LIN {X 0,Y 296.94,Z 400.103,A -85,B 0,C 180,E1 -15461.241,E2 -15461.241} C_VEL
LIN {X 0,Y 298.792,Z 385.556,A -85,B 0,C 180,E1 -15462.873,E2 -15462.873} C_VEL
LIN {X 0,Y 295.026,Z 372.369,A -85,B 0,C 180,E1 -15465.675,E2 -15465.675} C_VEL
LIN {X 0,Y 290.73,Z 360.298,A -85,B 0,C 180,E1 -15468.694,E2 -15468.694} C_VEL
LIN {X 0,Y 286.134,Z 349.446,A -85,B 0,C 180,E1 -15471.964,E2 -15471.964} C_VEL
LIN {X 0,Y 282.035,Z 341.18,A -85,B 0,C 180,E1 -15474.962,E2 -15474.962} C_VEL
LIN {X 0,Y 279.846,Z 337.032,A -85,B 0,C 180,E1 -15476.722,E2 -15476.722} C_VEL
LIN {X 0,Y 277.551,Z 332.713,A -85,B 0,C 180,E1 -15478.761,E2 -15478.761} C_VEL
LIN {X 0,Y 275.306,Z 328.719,A -85,B 0,C 180,E1 -15480.832,E2 -15480.832} C_VEL
LIN {X 0,Y 272.385,Z 324.11,A -85,B 0,C 180,E1 -15483.999,E2 -15483.999} C_VEL
LIN {X 0,Y 271.755,Z 322.71,A -85,B 0,C 180,E1 -15484.854,E2 -15484.854} C_VEL
LIN {X 0,Y 268.885,Z 319.004,A -85,B 0,C 180,E1 -15488.984,E2 -15488.984} C_VEL
LIN {X 0,Y 268.106,Z 317.079,A -85,B 0,C 180,E1 -15490.964,E2 -15490.964} C_VEL
LIN {X 0,Y 266.633,Z 315.935,A -85,B 0,C 180,E1 -15497.024,E2 -15497.024} C_VEL
LIN {X 0,Y 267.959,Z 316.873,A -85,B 0,C 180,E1 -15502.891,E2 -15502.891} C_VEL
LIN {X 0,Y 268.11,Z 322.342,A -85,B 0,C 180,E1 -15505.632,E2 -15505.632} C_VEL
LIN {X 0,Y 268.563,Z 325.134,A -85,B 0,C 180,E1 -15506.834,E2 -15506.834} C_VEL
LIN {X 0,Y 280.399,Z 343.647,A -85,B 0,C 180,E1 -15510.42,E2 -15510.42} C_VEL
LIN {X 0,Y 293.861,Z 366.106,A -85,B 0,C 180,E1 -15514.094,E2 -15514.094} C_VEL
LIN {X 0,Y 307.067,Z 389.595,A -85,B 0,C 180,E1 -15517.363,E2 -15517.363} C_VEL
LIN {X 0,Y 311.122,Z 397.45,A -85,B 0,C 180,E1 -15518.324,E2 -15518.324} C_VEL
LIN {X 0,Y 295.469,Z 576.065,A -85,B 0,C 180,E1 -15523.892,E2 -15523.892} C_VEL
LIN {X 0,Y 292.753,Z 597.216,A -85,B 0,C 180,E1 -15524.876,E2 -15524.876} C_VEL
LIN {X 0,Y 289.439,Z 617.893,A -85,B 0,C 180,E1 -15526.18,E2 -15526.18} C_VEL
LIN {X 0,Y 285.489,Z 638.664,A -85,B 0,C 180,E1 -15527.884,E2 -15527.884} C_VEL
LIN {X 0,Y 281.43,Z 657.558,A -85,B 0,C 180,E1 -15529.832,E2 -15529.832} C_VEL
LIN {X 0,Y 277.005,Z 676.334,A -85,B 0,C 180,E1 -15532.23,E2 -15532.23} C_VEL
LIN {X 0,Y 272.656,Z 693.714,A -85,B 0,C 180,E1 -15534.957,E2 -15534.957} C_VEL
LIN {X 0,Y 268.576,Z 709.476,A -85,B 0,C 180,E1 -15537.964,E2 -15537.964} C_VEL
LIN {X 0,Y 264.829,Z 724.067,A -85,B 0,C 180,E1 -15541.351,E2 -15541.351} C_VEL
LIN {X 0,Y 261.74,Z 736.697,A -85,B 0,C 180,E1 -15544.914,E2 -15544.914} C_VEL
LIN {X 0,Y 259.298,Z 747.805,A -85,B 0,C 180,E1 -15548.751,E2 -15548.751} C_VEL
LIN {X 0,Y 257.574,Z 757.323,A -85,B 0,C 180,E1 -15552.844,E2 -15552.844} C_VEL
LIN {X 0,Y 256.562,Z 766.176,A -85,B 0,C 180,E1 -15557.168,E2 -15557.168} C_VEL
LIN {X 0,Y 256.224,Z 771.289,A -85,B 0,C 180,E1 -15560.57,E2 -15560.57} C_VEL
LIN {X 0,Y 256.172,Z 774.841,A -85,B 0,C 180,E1 -15564.178,E2 -15564.178} C_VEL
LIN {X 0,Y 256.225,Z 776.542,A -85,B 0,C 180,E1 -15567.542,E2 -15567.542} C_VEL
LIN {X 0,Y 256.224,Z 776.895,A -85,B 0,C 180,E1 -15571.791,E2 -15571.791} C_VEL
LIN {X 0,Y 256.095,Z 776.47,A -85,B 0,C 180,E1 -15575.604,E2 -15575.604} C_VEL
LIN {X 0,Y 256.135,Z 774.535,A -85,B 0,C 180,E1 -15579.666,E2 -15579.666} C_VEL
LIN {X 0,Y 256.782,Z 770.746,A -85,B 0,C 180,E1 -15584.177,E2 -15584.177} C_VEL
LIN {X 0,Y 258.426,Z 765.131,A -85,B 0,C 180,E1 -15588.734,E2 -15588.734} C_VEL
LIN {X 0,Y 261.437,Z 757.306,A -85,B 0,C 180,E1 -15593.44,E2 -15593.44} C_VEL
LIN {X 0,Y 265.948,Z 747.434,A -85,B 0,C 180,E1 -15598.033,E2 -15598.033} C_VEL
LIN {X 0,Y 272.081,Z 735.449,A -85,B 0,C 180,E1 -15602.45,E2 -15602.45} C_VEL
LIN {X 0,Y 279.493,Z 722.038,A -85,B 0,C 180,E1 -15606.433,E2 -15606.433} C_VEL
LIN {X 0,Y 288.993,Z 705.853,A -85,B 0,C 180,E1 -15610.317,E2 -15610.317} C_VEL
LIN {X 0,Y 299.761,Z 688.525,A -85,B 0,C 180,E1 -15613.668,E2 -15613.668} C_VEL
LIN {X 0,Y 311.664,Z 670.423,A -85,B 0,C 180,E1 -15616.474,E2 -15616.474} C_VEL
LIN {X 0,Y 316.699,Z 662.999,A -85,B 0,C 180,E1 -15617.467,E2 -15617.467} C_VEL
LIN {X 0,Y 304.303,Z 679.759,A -85,B 0,C 180,E1 -15620.155,E2 -15620.155} C_VEL
LIN {X 0,Y 293.114,Z 695.355,A -85,B 0,C 180,E1 -15623.349,E2 -15623.349} C_VEL
LIN {X 0,Y 283.18,Z 709.698,A -85,B 0,C 180,E1 -15627.062,E2 -15627.062} C_VEL
LIN {X 0,Y 275.344,Z 721.405,A -85,B 0,C 180,E1 -15630.884,E2 -15630.884} C_VEL
LIN {X 0,Y 269.011,Z 731.149,A -85,B 0,C 180,E1 -15634.931,E2 -15634.931} C_VEL
LIN {X 0,Y 264.108,Z 738.947,A -85,B 0,C 180,E1 -15639.154,E2 -15639.154} C_VEL
LIN {X 0,Y 260.554,Z 744.818,A -85,B 0,C 180,E1 -15643.503,E2 -15643.503} C_VEL
LIN {X 0,Y 258.222,Z 748.792,A -85,B 0,C 180,E1 -15647.932,E2 -15647.932} C_VEL
LIN {X 0,Y 256.91,Z 750.895,A -85,B 0,C 180,E1 -15652.397,E2 -15652.397} C_VEL
LIN {X 0,Y 256.377,Z 751.195,A -85,B 0,C 180,E1 -15656.423,E2 -15656.423} C_VEL
LIN {X 0,Y 256.196,Z 749.887,A -85,B 0,C 180,E1 -15660.448,E2 -15660.448} C_VEL
LIN {X 0,Y 256.191,Z 747.15,A -85,B 0,C 180,E1 -15664.253,E2 -15664.253} C_VEL
LIN {X 0,Y 256.434,Z 742.885,A -85,B 0,C 180,E1 -15668.07,E2 -15668.07} C_VEL
LIN {X 0,Y 257.125,Z 736.57,A -85,B 0,C 180,E1 -15672.122,E2 -15672.122} C_VEL
LIN {X 0,Y 258.365,Z 728.743,A -85,B 0,C 180,E1 -15675.949,E2 -15675.949} C_VEL
LIN {X 0,Y 260.321,Z 718.846,A -85,B 0,C 180,E1 -15679.773,E2 -15679.773} C_VEL
LIN {X 0,Y 262.858,Z 707.504,A -85,B 0,C 180,E1 -15683.304,E2 -15683.304} C_VEL
LIN {X 0,Y 265.921,Z 694.644,A -85,B 0,C 180,E1 -15686.58,E2 -15686.58} C_VEL
LIN {X 0,Y 269.39,Z 680.327,A -85,B 0,C 180,E1 -15689.581,E2 -15689.581} C_VEL
LIN {X 0,Y 273.303,Z 663.874,A -85,B 0,C 180,E1 -15692.41,E2 -15692.41} C_VEL
LIN {X 0,Y 277.26,Z 646.249,A -85,B 0,C 180,E1 -15694.862,E2 -15694.862} C_VEL
LIN {X 0,Y 281.09,Z 627.597,A -85,B 0,C 180,E1 -15696.953,E2 -15696.953} C_VEL
LIN {X 0,Y 284.671,Z 608.006,A -85,B 0,C 180,E1 -15698.698,E2 -15698.698} C_VEL
LIN {X 0,Y 287.862,Z 587.393,A -85,B 0,C 180,E1 -15700.115,E2 -15700.115} C_VEL
LIN {X 0,Y 290.507,Z 566.391,A -85,B 0,C 180,E1 -15701.175,E2 -15701.175} C_VEL
LIN {X 0,Y 299.392,Z 466.167,A -85,B 0,C 180,E1 -15704.569,E2 -15704.569} C_VEL
LIN {X 0,Y 305.766,Z 396.925,A -85,B 0,C 180,E1 -15706.789,E2 -15706.789} C_VEL
LIN {X 0,Y 293.128,Z 372.457,A -85,B 0,C 180,E1 -15709.952,E2 -15709.952} C_VEL
LIN {X 0,Y 281.063,Z 350.849,A -85,B 0,C 180,E1 -15713.233,E2 -15713.233} C_VEL
LIN {X 0,Y 272.665,Z 336.54,A -85,B 0,C 180,E1 -15715.742,E2 -15715.742} C_VEL
LIN {X 0,Y 271.176,Z 332.651,A -85,B 0,C 180,E1 -15716.965,E2 -15716.965} C_VEL
LIN {X 0,Y 272.605,Z 332.766,A -85,B 0,C 180,E1 -15717.523,E2 -15717.523} C_VEL
LIN {X 0,Y 273.848,Z 333.25,A -85,B 0,C 180,E1 -15717.896,E2 -15717.896} C_VEL
LIN {X 0,Y 279.927,Z 346.608,A -85,B 0,C 180,E1 -15721.25,E2 -15721.25} C_VEL
LIN {X 0,Y 286.015,Z 361.966,A -85,B 0,C 180,E1 -15724.642,E2 -15724.642} C_VEL
LIN {X 0,Y 291.59,Z 378.781,A -85,B 0,C 180,E1 -15727.934,E2 -15727.934} C_VEL
LIN {X 0,Y 292.582,Z 382.952,A -85,B 0,C 180,E1 -15728.655,E2 -15728.655} C_VEL
LIN {X 0,Y 287.272,Z 425.798,A -85,B 0,C 180,E1 -15733.415,E2 -15733.415} C_VEL
LIN {X 0,Y 281.887,Z 470.765,A -85,B 0,C 180,E1 -15738.437,E2 -15738.437} C_VEL
LIN {X 0,Y 280.377,Z 484.638,A -85,B 0,C 180,E1 -15739.986,E2 -15739.986} C_VEL
LIN {X 0,Y 282.331,Z 509.846,A -85,B 0,C 180,E1 -15741.017,E2 -15741.017} C_VEL
LIN {X 0,Y 277.427,Z 629.056,A -85,B 0,C 180,E1 -15744.096,E2 -15744.096} C_VEL
LIN {X 0,Y 276.177,Z 645.328,A -85,B 0,C 180,E1 -15744.896,E2 -15744.896} C_VEL
LIN {X 0,Y 274.405,Z 660.879,A -85,B 0,C 180,E1 -15746.028,E2 -15746.028} C_VEL
LIN {X 0,Y 272.222,Z 675.36,A -85,B 0,C 180,E1 -15747.472,E2 -15747.472} C_VEL
LIN {X 0,Y 269.588,Z 689.834,A -85,B 0,C 180,E1 -15749.36,E2 -15749.36} C_VEL
LIN {X 0,Y 266.915,Z 702.546,A -85,B 0,C 180,E1 -15751.5,E2 -15751.5} C_VEL
LIN {X 0,Y 264.139,Z 714.779,A -85,B 0,C 180,E1 -15754.122,E2 -15754.122} C_VEL
LIN {X 0,Y 261.785,Z 724.548,A -85,B 0,C 180,E1 -15756.797,E2 -15756.797} C_VEL
LIN {X 0,Y 259.615,Z 733.633,A -85,B 0,C 180,E1 -15759.978,E2 -15759.978} C_VEL
LIN {X 0,Y 258.037,Z 740.606,A -85,B 0,C 180,E1 -15763.213,E2 -15763.213} C_VEL
LIN {X 0,Y 256.943,Z 746.215,A -85,B 0,C 180,E1 -15766.806,E2 -15766.806} C_VEL
LIN {X 0,Y 256.412,Z 749.748,A -85,B 0,C 180,E1 -15770.304,E2 -15770.304} C_VEL
LIN {X 0,Y 256.231,Z 751.673,A -85,B 0,C 180,E1 -15774.059,E2 -15774.059} C_VEL
LIN {X 0,Y 256.302,Z 751.729,A -85,B 0,C 180,E1 -15777.657,E2 -15777.657} C_VEL
LIN {X 0,Y 256.718,Z 749.922,A -85,B 0,C 180,E1 -15781.464,E2 -15781.464} C_VEL
LIN {X 0,Y 257.406,Z 747.146,A -85,B 0,C 180,E1 -15784.411,E2 -15784.411} C_VEL
LIN {X 0,Y 256.996,Z 745.207,A -85,B 0,C 180,E1 -15786.083,E2 -15786.083} C_VEL
LIN {X 0,Y 253.978,Z 740.913,A -85,B 0,C 180,E1 -15789.129,E2 -15789.129} C_VEL
LIN {X 0,Y 252.927,Z 737.614,A -85,B 0,C 180,E1 -15790.989,E2 -15790.989} C_VEL
LIN {X 0,Y 253.22,Z 735.69,A -85,B 0,C 180,E1 -15791.898,E2 -15791.898} C_VEL
LIN {X 0,Y 255.85,Z 727.502,A -85,B 0,C 180,E1 -15795.015,E2 -15795.015} C_VEL
LIN {X 0,Y 258.986,Z 717.445,A -85,B 0,C 180,E1 -15797.966,E2 -15797.966} C_VEL
LIN {X 0,Y 262.25,Z 706.223,A -85,B 0,C 180,E1 -15800.534,E2 -15800.534} C_VEL
LIN {X 0,Y 265.744,Z 692.935,A -85,B 0,C 180,E1 -15802.901,E2 -15802.901} C_VEL
LIN {X 0,Y 268.866,Z 679.065,A -85,B 0,C 180,E1 -15804.8,E2 -15804.8} C_VEL
LIN {X 0,Y 271.687,Z 663.938,A -85,B 0,C 180,E1 -15806.376,E2 -15806.376} C_VEL
LIN {X 0,Y 273.868,Z 648.202,A -85,B 0,C 180,E1 -15807.563,E2 -15807.563} C_VEL
LIN {X 0,Y 275.419,Z 631.651,A -85,B 0,C 180,E1 -15808.411,E2 -15808.411} C_VEL
LIN {X 0,Y 278.117,Z 576.528,A -85,B 0,C 180,E1 -15809.917,E2 -15809.917} C_VEL
LIN {X 0,Y 281.382,Z 509.252,A -85,B 0,C 180,E1 -15811.687,E2 -15811.687} C_VEL
LIN {X 0,Y 279.555,Z 485.416,A -85,B 0,C 180,E1 -15812.939,E2 -15812.939} C_VEL
LIN {X 0,Y 285.902,Z 439.143,A -85,B 0,C 180,E1 -15818.132,E2 -15818.132} C_VEL
LIN {X 0,Y 292.228,Z 395.584,A -85,B 0,C 180,E1 -15822.989,E2 -15822.989} C_VEL
LIN {X 0,Y 293.049,Z 389.555,A -85,B 0,C 180,E1 -15823.65,E2 -15823.65} C_VEL
LIN {X 0,Y 289.558,Z 376.947,A -85,B 0,C 180,E1 -15826.419,E2 -15826.419} C_VEL
LIN {X 0,Y 285.465,Z 365.026,A -85,B 0,C 180,E1 -15829.505,E2 -15829.505} C_VEL
LIN {X 0,Y 281.342,Z 355.057,A -85,B 0,C 180,E1 -15832.649,E2 -15832.649} C_VEL
LIN {X 0,Y 277.52,Z 347.06,A -85,B 0,C 180,E1 -15835.66,E2 -15835.66} C_VEL
LIN {X 0,Y 275.656,Z 343.37,A -85,B 0,C 180,E1 -15837.297,E2 -15837.297} C_VEL
LIN {X 0,Y 273.619,Z 339.446,A -85,B 0,C 180,E1 -15839.162,E2 -15839.162} C_VEL
LIN {X 0,Y 271.208,Z 334.904,A -85,B 0,C 180,E1 -15841.689,E2 -15841.689} C_VEL
LIN {X 0,Y 269.01,Z 331.316,A -85,B 0,C 180,E1 -15844.262,E2 -15844.262} C_VEL
LIN {X 0,Y 268.402,Z 329.91,A -85,B 0,C 180,E1 -15845.129,E2 -15845.129} C_VEL
LIN {X 0,Y 265.797,Z 326.228,A -85,B 0,C 180,E1 -15849.308,E2 -15849.308} C_VEL
LIN {X 0,Y 265.181,Z 324.503,A -85,B 0,C 180,E1 -15851.086,E2 -15851.086} C_VEL
LIN {X 0,Y 263.927,Z 323.468,A -85,B 0,C 180,E1 -15857.186,E2 -15857.186} C_VEL
LIN {X 0,Y 265.171,Z 324.337,A -85,B 0,C 180,E1 -15862.519,E2 -15862.519} C_VEL
LIN {X 0,Y 265.167,Z 329.151,A -85,B 0,C 180,E1 -15864.98,E2 -15864.98} C_VEL
LIN {X 0,Y 265.422,Z 332.988,A -85,B 0,C 180,E1 -15866.572,E2 -15866.572} C_VEL
LIN {X 0,Y 277.388,Z 352.176,A -85,B 0,C 180,E1 -15870.306,E2 -15870.306} C_VEL
LIN {X 0,Y 291.163,Z 375.535,A -85,B 0,C 180,E1 -15874.097,E2 -15874.097} C_VEL
LIN {X 0,Y 304.653,Z 399.967,A -85,B 0,C 180,E1 -15877.456,E2 -15877.456} C_VEL
LIN {X 0,Y 288.575,Z 575.961,A -85,B 0,C 180,E1 -15883.096,E2 -15883.096} C_VEL
LIN {X 0,Y 285.646,Z 597.916,A -85,B 0,C 180,E1 -15884.15,E2 -15884.15} C_VEL
LIN {X 0,Y 282.271,Z 618.214,A -85,B 0,C 180,E1 -15885.468,E2 -15885.468} C_VEL
LIN {X 0,Y 278.195,Z 638.944,A -85,B 0,C 180,E1 -15887.216,E2 -15887.216} C_VEL
LIN {X 0,Y 274,Z 657.836,A -85,B 0,C 180,E1 -15889.221,E2 -15889.221} C_VEL
LIN {X 0,Y 269.634,Z 675.826,A -85,B 0,C 180,E1 -15891.573,E2 -15891.573} C_VEL
LIN {X 0,Y 265.139,Z 693.255,A -85,B 0,C 180,E1 -15894.368,E2 -15894.368} C_VEL
LIN {X 0,Y 260.913,Z 709.095,A -85,B 0,C 180,E1 -15897.465,E2 -15897.465} C_VEL
LIN {X 0,Y 257.077,Z 723.582,A -85,B 0,C 180,E1 -15900.914,E2 -15900.914} C_VEL
LIN {X 0,Y 253.884,Z 736.239,A -85,B 0,C 180,E1 -15904.582,E2 -15904.582} C_VEL
LIN {X 0,Y 251.35,Z 747.43,A -85,B 0,C 180,E1 -15908.565,E2 -15908.565} C_VEL
LIN {X 0,Y 249.316,Z 760.034,A -85,B 0,C 180,E1 -15913.699,E2 -15913.699} C_VEL
LIN {X 0,Y 248.554,Z 766.708,A -85,B 0,C 180,E1 -15917.22,E2 -15917.22} C_VEL
LIN {X 0,Y 248.207,Z 771.783,A -85,B 0,C 180,E1 -15920.964,E2 -15920.964} C_VEL
LIN {X 0,Y 248.173,Z 774.842,A -85,B 0,C 180,E1 -15924.454,E2 -15924.454} C_VEL
LIN {X 0,Y 248.24,Z 776.268,A -85,B 0,C 180,E1 -15927.925,E2 -15927.925} C_VEL
LIN {X 0,Y 248.223,Z 776.367,A -85,B 0,C 180,E1 -15932.311,E2 -15932.311} C_VEL
LIN {X 0,Y 248.094,Z 775.911,A -85,B 0,C 180,E1 -15936.249,E2 -15936.249} C_VEL
LIN {X 0,Y 248.218,Z 773.809,A -85,B 0,C 180,E1 -15940.681,E2 -15940.681} C_VEL
LIN {X 0,Y 249.171,Z 769.632,A -85,B 0,C 180,E1 -15945.625,E2 -15945.625} C_VEL
LIN {X 0,Y 251.338,Z 763.593,A -85,B 0,C 180,E1 -15950.494,E2 -15950.494} C_VEL
LIN {X 0,Y 254.987,Z 755.598,A -85,B 0,C 180,E1 -15955.306,E2 -15955.306} C_VEL
LIN {X 0,Y 260.25,Z 745.641,A -85,B 0,C 180,E1 -15959.966,E2 -15959.966} C_VEL
LIN {X 0,Y 267.22,Z 733.705,A -85,B 0,C 180,E1 -15964.404,E2 -15964.404} C_VEL
LIN {X 0,Y 275.965,Z 719.805,A -85,B 0,C 180,E1 -15968.551,E2 -15968.551} C_VEL
LIN {X 0,Y 287.073,Z 703.228,A -85,B 0,C 180,E1 -15972.51,E2 -15972.51} C_VEL
LIN {X 0,Y 299.64,Z 685.661,A -85,B 0,C 180,E1 -15975.845,E2 -15975.845} C_VEL
LIN {X 0,Y 307.526,Z 675.142,A -85,B 0,C 180,E1 -15977.534,E2 -15977.534} C_VEL
LIN {X 0,Y 294.888,Z 690.385,A -85,B 0,C 180,E1 -15980.4,E2 -15980.4} C_VEL
LIN {X 0,Y 282.713,Z 705.662,A -85,B 0,C 180,E1 -15984.088,E2 -15984.088} C_VEL
LIN {X 0,Y 272.716,Z 718.764,A -85,B 0,C 180,E1 -15988.134,E2 -15988.134} C_VEL
LIN {X 0,Y 264.863,Z 729.274,A -85,B 0,C 180,E1 -15992.334,E2 -15992.334} C_VEL
LIN {X 0,Y 258.947,Z 737.428,A -85,B 0,C 180,E1 -15996.566,E2 -15996.566} C_VEL
LIN {X 0,Y 254.487,Z 743.76,A -85,B 0,C 180,E1 -16000.969,E2 -16000.969} C_VEL
LIN {X 0,Y 251.395,Z 748.261,A -85,B 0,C 180,E1 -16005.49,E2 -16005.49} C_VEL
LIN {X 0,Y 249.503,Z 750.937,A -85,B 0,C 180,E1 -16010.078,E2 -16010.078} C_VEL
LIN {X 0,Y 248.594,Z 751.782,A -85,B 0,C 180,E1 -16014.461,E2 -16014.461} C_VEL
LIN {X 0,Y 248.261,Z 751.006,A -85,B 0,C 180,E1 -16018.616,E2 -16018.616} C_VEL
LIN {X 0,Y 248.173,Z 748.831,A -85,B 0,C 180,E1 -16022.541,E2 -16022.541} C_VEL
LIN {X 0,Y 248.31,Z 744.859,A -85,B 0,C 180,E1 -16026.707,E2 -16026.707} C_VEL
LIN {X 0,Y 248.853,Z 739.068,A -85,B 0,C 180,E1 -16030.886,E2 -16030.886} C_VEL
LIN {X 0,Y 250.004,Z 731.303,A -85,B 0,C 180,E1 -16035.069,E2 -16035.069} C_VEL
LIN {X 0,Y 251.806,Z 721.935,A -85,B 0,C 180,E1 -16039.003,E2 -16039.003} C_VEL
LIN {X 0,Y 254.234,Z 711.077,A -85,B 0,C 180,E1 -16042.671,E2 -16042.671} C_VEL
LIN {X 0,Y 257.275,Z 698.511,A -85,B 0,C 180,E1 -16046.133,E2 -16046.133} C_VEL
LIN {X 0,Y 260.864,Z 684.098,A -85,B 0,C 180,E1 -16049.382,E2 -16049.382} C_VEL
LIN {X 0,Y 264.765,Z 668.262,A -85,B 0,C 180,E1 -16052.302,E2 -16052.302} C_VEL
LIN {X 0,Y 268.892,Z 650.709,A -85,B 0,C 180,E1 -16054.936,E2 -16054.936} C_VEL
LIN {X 0,Y 272.949,Z 632.099,A -85,B 0,C 180,E1 -16057.188,E2 -16057.188} C_VEL
LIN {X 0,Y 276.751,Z 612.591,A -85,B 0,C 180,E1 -16059.071,E2 -16059.071} C_VEL
LIN {X 0,Y 280.116,Z 592.33,A -85,B 0,C 180,E1 -16060.583,E2 -16060.583} C_VEL
LIN {X 0,Y 283.01,Z 571.163,A -85,B 0,C 180,E1 -16061.757,E2 -16061.757} C_VEL
LIN {X 0,Y 285.913,Z 541.776,A -85,B 0,C 180,E1 -16062.885,E2 -16062.885} C_VEL
LIN {X 0,Y 299.252,Z 399.79,A -85,B 0,C 180,E1 -16067.637,E2 -16067.637} C_VEL
LIN {X 0,Y 287.388,Z 376.669,A -85,B 0,C 180,E1 -16070.711,E2 -16070.711} C_VEL
LIN {X 0,Y 275.771,Z 355.743,A -85,B 0,C 180,E1 -16073.964,E2 -16073.964} C_VEL
LIN {X 0,Y 266.659,Z 340.131,A -85,B 0,C 180,E1 -16076.806,E2 -16076.806} C_VEL
LIN {X 0,Y 266.891,Z 339.624,A -85,B 0,C 180,E1 -16077.154,E2 -16077.154} C_VEL
LIN {X 0,Y 268.978,Z 339.864,A -85,B 0,C 180,E1 -16077.746,E2 -16077.746} C_VEL
LIN {X 0,Y 275.266,Z 354.159,A -85,B 0,C 180,E1 -16081.347,E2 -16081.347} C_VEL
LIN {X 0,Y 281.019,Z 369.487,A -85,B 0,C 180,E1 -16084.723,E2 -16084.723} C_VEL
LIN {X 0,Y 285.974,Z 385.172,A -85,B 0,C 180,E1 -16087.813,E2 -16087.813} C_VEL
LIN {X 0,Y 281.647,Z 419.515,A -85,B 0,C 180,E1 -16091.687,E2 -16091.687} C_VEL
LIN {X 0,Y 275.942,Z 464.782,A -85,B 0,C 180,E1 -16096.802,E2 -16096.802} C_VEL
LIN {X 0,Y 273.579,Z 484.324,A -85,B 0,C 180,E1 -16099.042,E2 -16099.042} C_VEL
LIN {X 0,Y 275.499,Z 510.719,A -85,B 0,C 180,E1 -16100.17,E2 -16100.17} C_VEL
LIN {X 0,Y 270.405,Z 629.316,A -85,B 0,C 180,E1 -16103.296,E2 -16103.296} C_VEL
LIN {X 0,Y 269.114,Z 645.535,A -85,B 0,C 180,E1 -16104.107,E2 -16104.107} C_VEL
LIN {X 0,Y 267.249,Z 661.287,A -85,B 0,C 180,E1 -16105.276,E2 -16105.276} C_VEL
LIN {X 0,Y 264.975,Z 675.763,A -85,B 0,C 180,E1 -16106.753,E2 -16106.753} C_VEL
LIN {X 0,Y 262.231,Z 690.238,A -85,B 0,C 180,E1 -16108.687,E2 -16108.687} C_VEL
LIN {X 0,Y 259.442,Z 702.948,A -85,B 0,C 180,E1 -16110.881,E2 -16110.881} C_VEL
LIN {X 0,Y 256.54,Z 715.184,A -85,B 0,C 180,E1 -16113.573,E2 -16113.573} C_VEL
LIN {X 0,Y 253.89,Z 725.671,A -85,B 0,C 180,E1 -16116.555,E2 -16116.555} C_VEL
LIN {X 0,Y 251.798,Z 734.038,A -85,B 0,C 180,E1 -16119.598,E2 -16119.598} C_VEL
LIN {X 0,Y 250.137,Z 741.007,A -85,B 0,C 180,E1 -16122.932,E2 -16122.932} C_VEL
LIN {X 0,Y 249.001,Z 746.517,A -85,B 0,C 180,E1 -16126.562,E2 -16126.562} C_VEL
LIN {X 0,Y 248.451,Z 749.972,A -85,B 0,C 180,E1 -16130,E2 -16130} C_VEL
LIN {X 0,Y 248.243,Z 751.951,A -85,B 0,C 180,E1 -16133.749,E2 -16133.749} C_VEL
LIN {X 0,Y 248.296,Z 752.234,A -85,B 0,C 180,E1 -16137.324,E2 -16137.324} C_VEL
LIN {X 0,Y 248.669,Z 750.756,A -85,B 0,C 180,E1 -16141.079,E2 -16141.079} C_VEL
LIN {X 0,Y 249.585,Z 747.388,A -85,B 0,C 180,E1 -16144.947,E2 -16144.947} C_VEL
LIN {X 0,Y 251.035,Z 742.53,A -85,B 0,C 180,E1 -16148.41,E2 -16148.41} C_VEL
LIN {X 0,Y 253.22,Z 735.69,A -85,B 0,C 180,E1 -16151.898,E2 -16151.898} C_VEL
LIN {X 0,Y 253.462,Z 732.181,A -85,B 0,C 180,E1 -16153.464,E2 -16153.464} C_VEL
LIN {X 0,Y 251.407,Z 724.108,A -85,B 0,C 180,E1 -16156.77,E2 -16156.77} C_VEL
LIN {X 0,Y 251.346,Z 719.743,A -85,B 0,C 180,E1 -16158.237,E2 -16158.237} C_VEL
LIN {X 0,Y 251.845,Z 717.662,A -85,B 0,C 180,E1 -16158.823,E2 -16158.823} C_VEL
LIN {X 0,Y 255.273,Z 706.473,A -85,B 0,C 180,E1 -16161.432,E2 -16161.432} C_VEL
LIN {X 0,Y 258.898,Z 693.357,A -85,B 0,C 180,E1 -16163.814,E2 -16163.814} C_VEL
LIN {X 0,Y 262.043,Z 680.108,A -85,B 0,C 180,E1 -16165.674,E2 -16165.674} C_VEL
LIN {X 0,Y 264.995,Z 665.102,A -85,B 0,C 180,E1 -16167.283,E2 -16167.283} C_VEL
LIN {X 0,Y 267.294,Z 649.691,A -85,B 0,C 180,E1 -16168.495,E2 -16168.495} C_VEL
LIN {X 0,Y 268.986,Z 632.949,A -85,B 0,C 180,E1 -16169.39,E2 -16169.39} C_VEL
LIN {X 0,Y 270.617,Z 602.218,A -85,B 0,C 180,E1 -16170.292,E2 -16170.292} C_VEL
LIN {X 0,Y 275.313,Z 510.209,A -85,B 0,C 180,E1 -16172.752,E2 -16172.752} C_VEL
LIN {X 0,Y 273.512,Z 485.979,A -85,B 0,C 180,E1 -16174.058,E2 -16174.058} C_VEL
LIN {X 0,Y 280.045,Z 440.73,A -85,B 0,C 180,E1 -16179.191,E2 -16179.191} C_VEL
LIN {X 0,Y 286.282,Z 399.532,A -85,B 0,C 180,E1 -16183.823,E2 -16183.823} C_VEL
LIN {X 0,Y 287.247,Z 393.097,A -85,B 0,C 180,E1 -16184.556,E2 -16184.556} C_VEL
LIN {X 0,Y 283.992,Z 380.77,A -85,B 0,C 180,E1 -16187.391,E2 -16187.391} C_VEL
LIN {X 0,Y 280.11,Z 369.196,A -85,B 0,C 180,E1 -16190.549,E2 -16190.549} C_VEL
LIN {X 0,Y 275.927,Z 358.91,A -85,B 0,C 180,E1 -16193.967,E2 -16193.967} C_VEL
LIN {X 0,Y 272.236,Z 350.875,A -85,B 0,C 180,E1 -16197.263,E2 -16197.263} C_VEL
LIN {X 0,Y 269.55,Z 345.877,A -85,B 0,C 180,E1 -16199.787,E2 -16199.787} C_VEL
LIN {X 0,Y 267.534,Z 341.803,A -85,B 0,C 180,E1 -16202.141,E2 -16202.141} C_VEL
LIN {X 0,Y 265.369,Z 337.748,A -85,B 0,C 180,E1 -16204.971,E2 -16204.971} C_VEL
LIN {X 0,Y 264.4,Z 336.5,A -85,B 0,C 180,E1 -16206.295,E2 -16206.295} C_VEL
LIN {X 0,Y 262.185,Z 331.841,A -85,B 0,C 180,E1 -16211.437,E2 -16211.437} C_VEL
LIN {X 0,Y 261.185,Z 330.989,A -85,B 0,C 180,E1 -16217.373,E2 -16217.373} C_VEL
LIN {X 0,Y 262.323,Z 331.785,A -85,B 0,C 180,E1 -16222.168,E2 -16222.168} C_VEL
LIN {X 0,Y 262.258,Z 336.015,A -85,B 0,C 180,E1 -16224.338,E2 -16224.338} C_VEL
LIN {X 0,Y 262.325,Z 340.027,A -85,B 0,C 180,E1 -16225.996,E2 -16225.996} C_VEL
LIN {X 0,Y 262.766,Z 341.877,A -85,B 0,C 180,E1 -16226.588,E2 -16226.588} C_VEL
LIN {X 0,Y 275.605,Z 362.845,A -85,B 0,C 180,E1 -16230.554,E2 -16230.554} C_VEL
LIN {X 0,Y 288.747,Z 385.611,A -85,B 0,C 180,E1 -16234.182,E2 -16234.182} C_VEL
LIN {X 0,Y 298.163,Z 403.236,A -85,B 0,C 180,E1 -16236.594,E2 -16236.594} C_VEL
LIN {X 0,Y 281.724,Z 575.658,A -85,B 0,C 180,E1 -16242.265,E2 -16242.265} C_VEL
LIN {X 0,Y 278.71,Z 597.541,A -85,B 0,C 180,E1 -16243.339,E2 -16243.339} C_VEL
LIN {X 0,Y 275.124,Z 618.407,A -85,B 0,C 180,E1 -16244.729,E2 -16244.729} C_VEL
LIN {X 0,Y 270.941,Z 639.009,A -85,B 0,C 180,E1 -16246.513,E2 -16246.513} C_VEL
LIN {X 0,Y 266.524,Z 658.262,A -85,B 0,C 180,E1 -16248.615,E2 -16248.615} C_VEL
LIN {X 0,Y 261.89,Z 676.708,A -85,B 0,C 180,E1 -16251.112,E2 -16251.112} C_VEL
LIN {X 0,Y 257.448,Z 693.416,A -85,B 0,C 180,E1 -16253.882,E2 -16253.882} C_VEL
LIN {X 0,Y 253.07,Z 709.33,A -85,B 0,C 180,E1 -16257.098,E2 -16257.098} C_VEL
LIN {X 0,Y 249.3,Z 723.174,A -85,B 0,C 180,E1 -16260.494,E2 -16260.494} C_VEL
LIN {X 0,Y 246.038,Z 735.711,A -85,B 0,C 180,E1 -16264.229,E2 -16264.229} C_VEL
LIN {X 0,Y 243.824,Z 745.568,A -85,B 0,C 180,E1 -16267.585,E2 -16267.585} C_VEL
LIN {X 0,Y 242.235,Z 754.919,A -85,B 0,C 180,E1 -16270.972,E2 -16270.972} C_VEL
LIN {X 0,Y 241.07,Z 762.731,A -85,B 0,C 180,E1 -16274.609,E2 -16274.609} C_VEL
LIN {X 0,Y 240.415,Z 768.58,A -85,B 0,C 180,E1 -16278.244,E2 -16278.244} C_VEL
LIN {X 0,Y 240.179,Z 772.874,A -85,B 0,C 180,E1 -16282.107,E2 -16282.107} C_VEL
LIN {X 0,Y 240.196,Z 775.247,A -85,B 0,C 180,E1 -16285.706,E2 -16285.706} C_VEL
LIN {X 0,Y 240.275,Z 776.015,A -85,B 0,C 180,E1 -16289.287,E2 -16289.287} C_VEL
LIN {X 0,Y 240.208,Z 775.827,A -85,B 0,C 180,E1 -16293.104,E2 -16293.104} C_VEL
LIN {X 0,Y 240.081,Z 775.292,A -85,B 0,C 180,E1 -16297.18,E2 -16297.18} C_VEL
LIN {X 0,Y 240.332,Z 773.094,A -85,B 0,C 180,E1 -16301.765,E2 -16301.765} C_VEL
LIN {X 0,Y 241.568,Z 768.888,A -85,B 0,C 180,E1 -16306.844,E2 -16306.844} C_VEL
LIN {X 0,Y 244.168,Z 762.817,A -85,B 0,C 180,E1 -16311.881,E2 -16311.881} C_VEL
LIN {X 0,Y 248.363,Z 754.893,A -85,B 0,C 180,E1 -16316.803,E2 -16316.803} C_VEL
LIN {X 0,Y 254.275,Z 745.109,A -85,B 0,C 180,E1 -16321.535,E2 -16321.535} C_VEL
LIN {X 0,Y 262.379,Z 732.889,A -85,B 0,C 180,E1 -16326.207,E2 -16326.207} C_VEL
LIN {X 0,Y 272.493,Z 718.725,A -85,B 0,C 180,E1 -16330.504,E2 -16330.504} C_VEL
LIN {X 0,Y 285.244,Z 702.064,A -85,B 0,C 180,E1 -16334.514,E2 -16334.514} C_VEL
LIN {X 0,Y 298.345,Z 686.007,A -85,B 0,C 180,E1 -16337.582,E2 -16337.582} C_VEL
LIN {X 0,Y 285.435,Z 700.019,A -85,B 0,C 180,E1 -16340.653,E2 -16340.653} C_VEL
LIN {X 0,Y 273.446,Z 713.571,A -85,B 0,C 180,E1 -16344.453,E2 -16344.453} C_VEL
LIN {X 0,Y 263.45,Z 725.221,A -85,B 0,C 180,E1 -16348.672,E2 -16348.672} C_VEL
LIN {X 0,Y 255.57,Z 734.646,A -85,B 0,C 180,E1 -16353.129,E2 -16353.129} C_VEL
LIN {X 0,Y 249.47,Z 742.124,A -85,B 0,C 180,E1 -16357.869,E2 -16357.869} C_VEL
LIN {X 0,Y 245.302,Z 747.328,A -85,B 0,C 180,E1 -16362.52,E2 -16362.52} C_VEL
LIN {X 0,Y 242.619,Z 750.632,A -85,B 0,C 180,E1 -16367.143,E2 -16367.143} C_VEL
LIN {X 0,Y 241.057,Z 752.219,A -85,B 0,C 180,E1 -16371.894,E2 -16371.894} C_VEL
LIN {X 0,Y 240.395,Z 752.015,A -85,B 0,C 180,E1 -16376.424,E2 -16376.424} C_VEL
LIN {X 0,Y 240.2,Z 750.233,A -85,B 0,C 180,E1 -16380.716,E2 -16380.716} C_VEL
LIN {X 0,Y 240.21,Z 747.067,A -85,B 0,C 180,E1 -16384.776,E2 -16384.776} C_VEL
LIN {X 0,Y 240.52,Z 742.34,A -85,B 0,C 180,E1 -16388.849,E2 -16388.849} C_VEL
LIN {X 0,Y 241.371,Z 735.455,A -85,B 0,C 180,E1 -16393.17,E2 -16393.17} C_VEL
LIN {X 0,Y 242.857,Z 727.042,A -85,B 0,C 180,E1 -16397.244,E2 -16397.244} C_VEL
LIN {X 0,Y 244.974,Z 717.208,A -85,B 0,C 180,E1 -16401.05,E2 -16401.05} C_VEL
LIN {X 0,Y 247.871,Z 705.176,A -85,B 0,C 180,E1 -16404.82,E2 -16404.82} C_VEL
LIN {X 0,Y 251.297,Z 691.714,A -85,B 0,C 180,E1 -16408.261,E2 -16408.261} C_VEL
LIN {X 0,Y 255.157,Z 676.643,A -85,B 0,C 180,E1 -16411.412,E2 -16411.412} C_VEL
LIN {X 0,Y 259.477,Z 659.25,A -85,B 0,C 180,E1 -16414.37,E2 -16414.37} C_VEL
LIN {X 0,Y 263.643,Z 641.466,A -85,B 0,C 180,E1 -16416.814,E2 -16416.814} C_VEL
LIN {X 0,Y 267.756,Z 622.179,A -85,B 0,C 180,E1 -16418.945,E2 -16418.945} C_VEL
LIN {X 0,Y 271.494,Z 602.071,A -85,B 0,C 180,E1 -16420.683,E2 -16420.683} C_VEL
LIN {X 0,Y 274.769,Z 581.052,A -85,B 0,C 180,E1 -16422.064,E2 -16422.064} C_VEL
LIN {X 0,Y 277.472,Z 558.924,A -85,B 0,C 180,E1 -16423.104,E2 -16423.104} C_VEL
LIN {X 0,Y 292.736,Z 402.476,A -85,B 0,C 180,E1 -16428.531,E2 -16428.531} C_VEL
LIN {X 0,Y 280.402,Z 378.491,A -85,B 0,C 180,E1 -16431.844,E2 -16431.844} C_VEL
LIN {X 0,Y 268.661,Z 357.396,A -85,B 0,C 180,E1 -16435.289,E2 -16435.289} C_VEL
LIN {X 0,Y 263.05,Z 347.539,A -85,B 0,C 180,E1 -16437.145,E2 -16437.145} C_VEL
LIN {X 0,Y 263.382,Z 346.943,A -85,B 0,C 180,E1 -16437.435,E2 -16437.435} C_VEL
LIN {X 0,Y 264.367,Z 347.015,A -85,B 0,C 180,E1 -16437.726,E2 -16437.726} C_VEL
LIN {X 0,Y 270.486,Z 361.582,A -85,B 0,C 180,E1 -16441.395,E2 -16441.395} C_VEL
LIN {X 0,Y 276.098,Z 377.318,A -85,B 0,C 180,E1 -16444.872,E2 -16444.872} C_VEL
LIN {X 0,Y 279.437,Z 389.009,A -85,B 0,C 180,E1 -16447.154,E2 -16447.154} C_VEL
LIN {X 0,Y 273.666,Z 431.774,A -85,B 0,C 180,E1 -16452.015,E2 -16452.015} C_VEL
LIN {X 0,Y 267.938,Z 475.725,A -85,B 0,C 180,E1 -16457.06,E2 -16457.06} C_VEL
LIN {X 0,Y 266.869,Z 485.441,A -85,B 0,C 180,E1 -16458.147,E2 -16458.147} C_VEL
LIN {X 0,Y 268.738,Z 511.464,A -85,B 0,C 180,E1 -16459.277,E2 -16459.277} C_VEL
LIN {X 0,Y 263.4,Z 629.84,A -85,B 0,C 180,E1 -16462.473,E2 -16462.473} C_VEL
LIN {X 0,Y 262.031,Z 646.203,A -85,B 0,C 180,E1 -16463.314,E2 -16463.314} C_VEL
LIN {X 0,Y 260.134,Z 661.581,A -85,B 0,C 180,E1 -16464.484,E2 -16464.484} C_VEL
LIN {X 0,Y 257.767,Z 676.09,A -85,B 0,C 180,E1 -16465.994,E2 -16465.994} C_VEL
LIN {X 0,Y 254.908,Z 690.584,A -85,B 0,C 180,E1 -16467.975,E2 -16467.975} C_VEL
LIN {X 0,Y 251.971,Z 703.426,A -85,B 0,C 180,E1 -16470.248,E2 -16470.248} C_VEL
LIN {X 0,Y 248.964,Z 715.561,A -85,B 0,C 180,E1 -16472.99,E2 -16472.99} C_VEL
LIN {X 0,Y 246.29,Z 725.681,A -85,B 0,C 180,E1 -16475.934,E2 -16475.934} C_VEL
LIN {X 0,Y 243.991,Z 734.43,A -85,B 0,C 180,E1 -16479.194,E2 -16479.194} C_VEL
LIN {X 0,Y 242.244,Z 741.402,A -85,B 0,C 180,E1 -16482.633,E2 -16482.633} C_VEL
LIN {X 0,Y 241.046,Z 746.913,A -85,B 0,C 180,E1 -16486.381,E2 -16486.381} C_VEL
LIN {X 0,Y 240.46,Z 750.406,A -85,B 0,C 180,E1 -16489.99,E2 -16489.99} C_VEL
LIN {X 0,Y 240.251,Z 752.346,A -85,B 0,C 180,E1 -16493.806,E2 -16493.806} C_VEL
LIN {X 0,Y 240.321,Z 752.618,A -85,B 0,C 180,E1 -16497.599,E2 -16497.599} C_VEL
LIN {X 0,Y 240.756,Z 751.048,A -85,B 0,C 180,E1 -16501.549,E2 -16501.549} C_VEL
LIN {X 0,Y 241.757,Z 747.721,A -85,B 0,C 180,E1 -16505.435,E2 -16505.435} C_VEL
LIN {X 0,Y 243.459,Z 742.459,A -85,B 0,C 180,E1 -16509.228,E2 -16509.228} C_VEL
LIN {X 0,Y 245.836,Z 735.559,A -85,B 0,C 180,E1 -16512.778,E2 -16512.778} C_VEL
LIN {X 0,Y 248.868,Z 726.664,A -85,B 0,C 180,E1 -16516.158,E2 -16516.158} C_VEL
LIN {X 0,Y 251.845,Z 717.662,A -85,B 0,C 180,E1 -16518.823,E2 -16518.823} C_VEL
LIN {X 0,Y 252.569,Z 712.778,A -85,B 0,C 180,E1 -16520.187,E2 -16520.187} C_VEL
LIN {X 0,Y 251.472,Z 702.771,A -85,B 0,C 180,E1 -16522.915,E2 -16522.915} C_VEL
LIN {X 0,Y 251.596,Z 696.374,A -85,B 0,C 180,E1 -16524.323,E2 -16524.323} C_VEL
LIN {X 0,Y 252.14,Z 693.786,A -85,B 0,C 180,E1 -16524.782,E2 -16524.782} C_VEL
LIN {X 0,Y 255.515,Z 680.254,A -85,B 0,C 180,E1 -16526.716,E2 -16526.716} C_VEL
LIN {X 0,Y 258.516,Z 665.707,A -85,B 0,C 180,E1 -16528.303,E2 -16528.303} C_VEL
LIN {X 0,Y 260.934,Z 650.295,A -85,B 0,C 180,E1 -16529.54,E2 -16529.54} C_VEL
LIN {X 0,Y 262.727,Z 633.392,A -85,B 0,C 180,E1 -16530.46,E2 -16530.46} C_VEL
LIN {X 0,Y 264.426,Z 602.955,A -85,B 0,C 180,E1 -16531.369,E2 -16531.369} C_VEL
LIN {X 0,Y 269.357,Z 511.316,A -85,B 0,C 180,E1 -16533.859,E2 -16533.859} C_VEL
LIN {X 0,Y 267.623,Z 486.252,A -85,B 0,C 180,E1 -16535.263,E2 -16535.263} C_VEL
LIN {X 0,Y 274.663,Z 440.447,A -85,B 0,C 180,E1 -16540.525,E2 -16540.525} C_VEL
LIN {X 0,Y 281.678,Z 396.905,A -85,B 0,C 180,E1 -16545.481,E2 -16545.481} C_VEL
LIN {X 0,Y 278.503,Z 384.661,A -85,B 0,C 180,E1 -16548.401,E2 -16548.401} C_VEL
LIN {X 0,Y 275.112,Z 374.138,A -85,B 0,C 180,E1 -16551.43,E2 -16551.43} C_VEL
LIN {X 0,Y 271.329,Z 364.565,A -85,B 0,C 180,E1 -16554.713,E2 -16554.713} C_VEL
LIN {X 0,Y 268.101,Z 357.243,A -85,B 0,C 180,E1 -16557.862,E2 -16557.862} C_VEL
LIN {X 0,Y 265.809,Z 352.672,A -85,B 0,C 180,E1 -16560.215,E2 -16560.215} C_VEL
LIN {X 0,Y 264.137,Z 348.957,A -85,B 0,C 180,E1 -16562.386,E2 -16562.386} C_VEL
LIN {X 0,Y 262.032,Z 344.964,A -85,B 0,C 180,E1 -16565.254,E2 -16565.254} C_VEL
LIN {X 0,Y 261.21,Z 343.736,A -85,B 0,C 180,E1 -16566.593,E2 -16566.593} C_VEL
LIN {X 0,Y 259.249,Z 339.266,A -85,B 0,C 180,E1 -16571.605,E2 -16571.605} C_VEL
LIN {X 0,Y 258.446,Z 338.509,A -85,B 0,C 180,E1 -16577.563,E2 -16577.563} C_VEL
LIN {X 0,Y 259.489,Z 339.421,A -85,B 0,C 180,E1 -16581.947,E2 -16581.947} C_VEL
LIN {X 0,Y 259.379,Z 345.514,A -85,B 0,C 180,E1 -16584.845,E2 -16584.845} C_VEL
LIN {X 0,Y 259.573,Z 350.003,A -85,B 0,C 180,E1 -16586.385,E2 -16586.385} C_VEL
LIN {X 0,Y 271.338,Z 369.415,A -85,B 0,C 180,E1 -16590.075,E2 -16590.075} C_VEL
LIN {X 0,Y 283.805,Z 391.256,A -85,B 0,C 180,E1 -16593.611,E2 -16593.611} C_VEL
LIN {X 0,Y 291.694,Z 406.109,A -85,B 0,C 180,E1 -16595.695,E2 -16595.695} C_VEL
LIN {X 0,Y 274.876,Z 575.506,A -85,B 0,C 180,E1 -16601.413,E2 -16601.413} C_VEL
LIN {X 0,Y 271.832,Z 596.932,A -85,B 0,C 180,E1 -16602.487,E2 -16602.487} C_VEL
LIN {X 0,Y 268.025,Z 618.404,A -85,B 0,C 180,E1 -16603.951,E2 -16603.951} C_VEL
LIN {X 0,Y 263.729,Z 638.906,A -85,B 0,C 180,E1 -16605.77,E2 -16605.77} C_VEL
LIN {X 0,Y 259.299,Z 657.672,A -85,B 0,C 180,E1 -16607.864,E2 -16607.864} C_VEL
LIN {X 0,Y 254.654,Z 675.677,A -85,B 0,C 180,E1 -16610.344,E2 -16610.344} C_VEL
LIN {X 0,Y 249.995,Z 692.7,A -85,B 0,C 180,E1 -16613.221,E2 -16613.221} C_VEL
LIN {X 0,Y 245.488,Z 708.606,A -85,B 0,C 180,E1 -16616.507,E2 -16616.507} C_VEL
LIN {X 0,Y 241.388,Z 723.196,A -85,B 0,C 180,E1 -16620.198,E2 -16620.198} C_VEL
LIN {X 0,Y 238.102,Z 736.125,A -85,B 0,C 180,E1 -16623.979,E2 -16623.979} C_VEL
LIN {X 0,Y 235.984,Z 746.974,A -85,B 0,C 180,E1 -16627.324,E2 -16627.324} C_VEL
LIN {X 0,Y 234.301,Z 755.943,A -85,B 0,C 180,E1 -16630.82,E2 -16630.82} C_VEL
LIN {X 0,Y 233.077,Z 763.404,A -85,B 0,C 180,E1 -16634.578,E2 -16634.578} C_VEL
LIN {X 0,Y 232.378,Z 769.258,A -85,B 0,C 180,E1 -16638.587,E2 -16638.587} C_VEL
LIN {X 0,Y 232.172,Z 772.992,A -85,B 0,C 180,E1 -16642.331,E2 -16642.331} C_VEL
LIN {X 0,Y 232.21,Z 775.067,A -85,B 0,C 180,E1 -16646.052,E2 -16646.052} C_VEL
LIN {X 0,Y 232.292,Z 775.579,A -85,B 0,C 180,E1 -16649.756,E2 -16649.756} C_VEL
LIN {X 0,Y 232.233,Z 775.277,A -85,B 0,C 180,E1 -16652.964,E2 -16652.964} C_VEL
LIN {X 0,Y 232.091,Z 774.894,A -85,B 0,C 180,E1 -16657.18,E2 -16657.18} C_VEL
LIN {X 0,Y 232.348,Z 773.008,A -85,B 0,C 180,E1 -16661.923,E2 -16661.923} C_VEL
LIN {X 0,Y 233.577,Z 769.389,A -85,B 0,C 180,E1 -16666.925,E2 -16666.925} C_VEL
LIN {X 0,Y 236.446,Z 763.468,A -85,B 0,C 180,E1 -16672.372,E2 -16672.372} C_VEL
LIN {X 0,Y 241.157,Z 755.58,A -85,B 0,C 180,E1 -16677.671,E2 -16677.671} C_VEL
LIN {X 0,Y 248.196,Z 745.291,A -85,B 0,C 180,E1 -16682.949,E2 -16682.949} C_VEL
LIN {X 0,Y 257.447,Z 732.968,A -85,B 0,C 180,E1 -16687.855,E2 -16687.855} C_VEL
LIN {X 0,Y 269.502,Z 718.104,A -85,B 0,C 180,E1 -16692.474,E2 -16692.474} C_VEL
LIN {X 0,Y 283.352,Z 702.222,A -85,B 0,C 180,E1 -16696.337,E2 -16696.337} C_VEL
LIN {X 0,Y 289.035,Z 696.015,A -85,B 0,C 180,E1 -16697.647,E2 -16697.647} C_VEL
LIN {X 0,Y 275.346,Z 709.401,A -85,B 0,C 180,E1 -16701.083,E2 -16701.083} C_VEL
LIN {X 0,Y 263.037,Z 721.802,A -85,B 0,C 180,E1 -16705.238,E2 -16705.238} C_VEL
LIN {X 0,Y 252.946,Z 732.321,A -85,B 0,C 180,E1 -16709.868,E2 -16709.868} C_VEL
LIN {X 0,Y 245.312,Z 740.47,A -85,B 0,C 180,E1 -16714.662,E2 -16714.662} C_VEL
LIN {X 0,Y 239.818,Z 746.395,A -85,B 0,C 180,E1 -16719.5,E2 -16719.5} C_VEL
LIN {X 0,Y 236.002,Z 750.456,A -85,B 0,C 180,E1 -16724.52,E2 -16724.52} C_VEL
LIN {X 0,Y 233.765,Z 752.545,A -85,B 0,C 180,E1 -16729.403,E2 -16729.403} C_VEL
LIN {X 0,Y 232.675,Z 752.869,A -85,B 0,C 180,E1 -16734.081,E2 -16734.081} C_VEL
LIN {X 0,Y 232.274,Z 751.624,A -85,B 0,C 180,E1 -16738.521,E2 -16738.521} C_VEL
LIN {X 0,Y 232.176,Z 749.013,A -85,B 0,C 180,E1 -16742.716,E2 -16742.716} C_VEL
LIN {X 0,Y 232.325,Z 744.909,A -85,B 0,C 180,E1 -16746.922,E2 -16746.922} C_VEL
LIN {X 0,Y 232.887,Z 739.168,A -85,B 0,C 180,E1 -16751.141,E2 -16751.141} C_VEL
LIN {X 0,Y 234.051,Z 731.644,A -85,B 0,C 180,E1 -16755.36,E2 -16755.36} C_VEL
LIN {X 0,Y 235.982,Z 722.115,A -85,B 0,C 180,E1 -16759.557,E2 -16759.557} C_VEL
LIN {X 0,Y 238.593,Z 711.091,A -85,B 0,C 180,E1 -16763.461,E2 -16763.461} C_VEL
LIN {X 0,Y 241.789,Z 698.652,A -85,B 0,C 180,E1 -16767.058,E2 -16767.058} C_VEL
LIN {X 0,Y 245.586,Z 684.276,A -85,B 0,C 180,E1 -16770.457,E2 -16770.457} C_VEL
LIN {X 0,Y 249.754,Z 668.328,A -85,B 0,C 180,E1 -16773.537,E2 -16773.537} C_VEL
LIN {X 0,Y 254.158,Z 650.692,A -85,B 0,C 180,E1 -16776.305,E2 -16776.305} C_VEL
LIN {X 0,Y 258.477,Z 632.032,A -85,B 0,C 180,E1 -16778.663,E2 -16778.663} C_VEL
LIN {X 0,Y 262.541,Z 612.369,A -85,B 0,C 180,E1 -16780.636,E2 -16780.636} C_VEL
LIN {X 0,Y 266.041,Z 592.568,A -85,B 0,C 180,E1 -16782.179,E2 -16782.179} C_VEL
LIN {X 0,Y 269.162,Z 571.164,A -85,B 0,C 180,E1 -16783.421,E2 -16783.421} C_VEL
LIN {X 0,Y 272.248,Z 542.164,A -85,B 0,C 180,E1 -16784.592,E2 -16784.592} C_VEL
LIN {X 0,Y 286.213,Z 405.215,A -85,B 0,C 180,E1 -16789.439,E2 -16789.439} C_VEL
LIN {X 0,Y 274.152,Z 381.732,A -85,B 0,C 180,E1 -16792.804,E2 -16792.804} C_VEL
LIN {X 0,Y 263.313,Z 362.162,A -85,B 0,C 180,E1 -16796.1,E2 -16796.1} C_VEL
LIN {X 0,Y 259.462,Z 355.12,A -85,B 0,C 180,E1 -16797.456,E2 -16797.456} C_VEL
LIN {X 0,Y 259.948,Z 354.608,A -85,B 0,C 180,E1 -16797.803,E2 -16797.803} C_VEL
LIN {X 0,Y 265.947,Z 369.757,A -85,B 0,C 180,E1 -16801.614,E2 -16801.614} C_VEL
LIN {X 0,Y 270.932,Z 384.639,A -85,B 0,C 180,E1 -16804.885,E2 -16804.885} C_VEL
LIN {X 0,Y 272.965,Z 392.002,A -85,B 0,C 180,E1 -16806.34,E2 -16806.34} C_VEL
LIN {X 0,Y 267.1,Z 433.334,A -85,B 0,C 180,E1 -16811.105,E2 -16811.105} C_VEL
LIN {X 0,Y 261.43,Z 474.987,A -85,B 0,C 180,E1 -16815.942,E2 -16815.942} C_VEL
LIN {X 0,Y 260.198,Z 485.826,A -85,B 0,C 180,E1 -16817.164,E2 -16817.164} C_VEL
LIN {X 0,Y 262.028,Z 512.289,A -85,B 0,C 180,E1 -16818.344,E2 -16818.344} C_VEL
LIN {X 0,Y 256.451,Z 630.322,A -85,B 0,C 180,E1 -16821.605,E2 -16821.605} C_VEL
LIN {X 0,Y 255.011,Z 646.741,A -85,B 0,C 180,E1 -16822.471,E2 -16822.471} C_VEL
LIN {X 0,Y 253.07,Z 661.849,A -85,B 0,C 180,E1 -16823.646,E2 -16823.646} C_VEL
LIN {X 0,Y 250.605,Z 676.391,A -85,B 0,C 180,E1 -16825.191,E2 -16825.191} C_VEL
LIN {X 0,Y 247.624,Z 690.905,A -85,B 0,C 180,E1 -16827.22,E2 -16827.22} C_VEL
LIN {X 0,Y 244.589,Z 703.65,A -85,B 0,C 180,E1 -16829.529,E2 -16829.529} C_VEL
LIN {X 0,Y 241.413,Z 715.913,A -85,B 0,C 180,E1 -16832.371,E2 -16832.371} C_VEL
LIN {X 0,Y 238.505,Z 726.419,A -85,B 0,C 180,E1 -16835.53,E2 -16835.53} C_VEL
LIN {X 0,Y 236.196,Z 734.801,A -85,B 0,C 180,E1 -16838.763,E2 -16838.763} C_VEL
LIN {X 0,Y 234.356,Z 741.78,A -85,B 0,C 180,E1 -16842.314,E2 -16842.314} C_VEL
LIN {X 0,Y 233.093,Z 747.297,A -85,B 0,C 180,E1 -16846.187,E2 -16846.187} C_VEL
LIN {X 0,Y 232.482,Z 750.755,A -85,B 0,C 180,E1 -16849.859,E2 -16849.859} C_VEL
LIN {X 0,Y 232.258,Z 752.739,A -85,B 0,C 180,E1 -16853.867,E2 -16853.867} C_VEL
LIN {X 0,Y 232.336,Z 753.025,A -85,B 0,C 180,E1 -16857.692,E2 -16857.692} C_VEL
LIN {X 0,Y 232.802,Z 751.526,A -85,B 0,C 180,E1 -16861.744,E2 -16861.744} C_VEL
LIN {X 0,Y 233.903,Z 748.174,A -85,B 0,C 180,E1 -16865.844,E2 -16865.844} C_VEL
LIN {X 0,Y 235.607,Z 743.314,A -85,B 0,C 180,E1 -16869.532,E2 -16869.532} C_VEL
LIN {X 0,Y 238.092,Z 736.561,A -85,B 0,C 180,E1 -16873.193,E2 -16873.193} C_VEL
LIN {X 0,Y 241.11,Z 728.302,A -85,B 0,C 180,E1 -16876.523,E2 -16876.523} C_VEL
LIN {X 0,Y 244.661,Z 718.184,A -85,B 0,C 180,E1 -16879.647,E2 -16879.647} C_VEL
LIN {X 0,Y 248.154,Z 707.442,A -85,B 0,C 180,E1 -16882.233,E2 -16882.233} C_VEL
LIN {X 0,Y 251.913,Z 694.598,A -85,B 0,C 180,E1 -16884.645,E2 -16884.645} C_VEL
LIN {X 0,Y 252.14,Z 693.786,A -85,B 0,C 180,E1 -16884.782,E2 -16884.782} C_VEL
LIN {X 0,Y 252.943,Z 687.682,A -85,B 0,C 180,E1 -16885.858,E2 -16885.858} C_VEL
LIN {X 0,Y 251.847,Z 673.719,A -85,B 0,C 180,E1 -16888.384,E2 -16888.384} C_VEL
LIN {X 0,Y 252.061,Z 667.063,A -85,B 0,C 180,E1 -16889.289,E2 -16889.289} C_VEL
LIN {X 0,Y 252.375,Z 665.07,A -85,B 0,C 180,E1 -16889.497,E2 -16889.497} C_VEL
LIN {X 0,Y 254.891,Z 649.347,A -85,B 0,C 180,E1 -16890.743,E2 -16890.743} C_VEL
LIN {X 0,Y 256.676,Z 632.86,A -85,B 0,C 180,E1 -16891.631,E2 -16891.631} C_VEL
LIN {X 0,Y 260.161,Z 572.117,A -85,B 0,C 180,E1 -16893.376,E2 -16893.376} C_VEL
LIN {X 0,Y 263.538,Z 512.271,A -85,B 0,C 180,E1 -16895.032,E2 -16895.032} C_VEL
LIN {X 0,Y 261.859,Z 487.034,A -85,B 0,C 180,E1 -16896.483,E2 -16896.483} C_VEL
LIN {X 0,Y 269.118,Z 441.982,A -85,B 0,C 180,E1 -16901.702,E2 -16901.702} C_VEL
LIN {X 0,Y 276.117,Z 400.724,A -85,B 0,C 180,E1 -16906.439,E2 -16906.439} C_VEL
LIN {X 0,Y 273.39,Z 389.42,A -85,B 0,C 180,E1 -16909.249,E2 -16909.249} C_VEL
LIN {X 0,Y 270.594,Z 380.2,A -85,B 0,C 180,E1 -16911.98,E2 -16911.98} C_VEL
LIN {X 0,Y 267.148,Z 370.865,A -85,B 0,C 180,E1 -16915.276,E2 -16915.276} C_VEL
LIN {X 0,Y 264.039,Z 363.618,A -85,B 0,C 180,E1 -16918.48,E2 -16918.48} C_VEL
LIN {X 0,Y 262.156,Z 359.505,A -85,B 0,C 180,E1 -16920.655,E2 -16920.655} C_VEL
LIN {X 0,Y 260.523,Z 355.857,A -85,B 0,C 180,E1 -16922.859,E2 -16922.859} C_VEL
LIN {X 0,Y 258.425,Z 351.439,A -85,B 0,C 180,E1 -16926.218,E2 -16926.218} C_VEL
LIN {X 0,Y 256.516,Z 347.354,A -85,B 0,C 180,E1 -16930.827,E2 -16930.827} C_VEL
LIN {X 0,Y 256.252,Z 346.625,A -85,B 0,C 180,E1 -16932.163,E2 -16932.163} C_VEL
LIN {X 0,Y 255.772,Z 346.054,A -85,B 0,C 180,E1 -16937.752,E2 -16937.752} C_VEL
LIN {X 0,Y 256.678,Z 346.655,A -85,B 0,C 180,E1 -16941.479,E2 -16941.479} C_VEL
LIN {X 0,Y 256.428,Z 352.391,A -85,B 0,C 180,E1 -16944.167,E2 -16944.167} C_VEL
LIN {X 0,Y 256.52,Z 358.28,A -85,B 0,C 180,E1 -16946.225,E2 -16946.225} C_VEL
LIN {X 0,Y 268.181,Z 377.95,A -85,B 0,C 180,E1 -16949.941,E2 -16949.941} C_VEL
LIN {X 0,Y 280.331,Z 399.558,A -85,B 0,C 180,E1 -16953.427,E2 -16953.427} C_VEL
LIN {X 0,Y 285.231,Z 409.114,A -85,B 0,C 180,E1 -16954.772,E2 -16954.772} C_VEL
LIN {X 0,Y 268.013,Z 575.619,A -85,B 0,C 180,E1 -16960.546,E2 -16960.546} C_VEL
LIN {X 0,Y 264.884,Z 596.863,A -85,B 0,C 180,E1 -16961.64,E2 -16961.64} C_VEL
LIN {X 0,Y 260.978,Z 618.204,A -85,B 0,C 180,E1 -16963.131,E2 -16963.131} C_VEL
LIN {X 0,Y 256.566,Z 638.64,A -85,B 0,C 180,E1 -16964.987,E2 -16964.987} C_VEL
LIN {X 0,Y 251.791,Z 658.206,A -85,B 0,C 180,E1 -16967.235,E2 -16967.235} C_VEL
LIN {X 0,Y 247.008,Z 676.133,A -85,B 0,C 180,E1 -16969.791,E2 -16969.791} C_VEL
LIN {X 0,Y 242.353,Z 692.634,A -85,B 0,C 180,E1 -16972.669,E2 -16972.669} C_VEL
LIN {X 0,Y 237.684,Z 708.623,A -85,B 0,C 180,E1 -16976.082,E2 -16976.082} C_VEL
LIN {X 0,Y 233.255,Z 724.496,A -85,B 0,C 180,E1 -16980.111,E2 -16980.111} C_VEL
LIN {X 0,Y 230.681,Z 736.731,A -85,B 0,C 180,E1 -16983.236,E2 -16983.236} C_VEL
LIN {X 0,Y 228.298,Z 747.641,A -85,B 0,C 180,E1 -16986.789,E2 -16986.789} C_VEL
LIN {X 0,Y 226.476,Z 756.403,A -85,B 0,C 180,E1 -16990.399,E2 -16990.399} C_VEL
LIN {X 0,Y 225.149,Z 763.621,A -85,B 0,C 180,E1 -16994.286,E2 -16994.286} C_VEL
LIN {X 0,Y 224.392,Z 769.313,A -85,B 0,C 180,E1 -16998.436,E2 -16998.436} C_VEL
LIN {X 0,Y 224.168,Z 773.013,A -85,B 0,C 180,E1 -17002.571,E2 -17002.571} C_VEL
LIN {X 0,Y 224.224,Z 774.858,A -85,B 0,C 180,E1 -17006.424,E2 -17006.424} C_VEL
LIN {X 0,Y 224.304,Z 775.142,A -85,B 0,C 180,E1 -17010.258,E2 -17010.258} C_VEL
LIN {X 0,Y 224.239,Z 774.681,A -85,B 0,C 180,E1 -17013.326,E2 -17013.326} C_VEL
LIN {X 0,Y 224.104,Z 774.334,A -85,B 0,C 180,E1 -17017.953,E2 -17017.953} C_VEL
LIN {X 0,Y 224.526,Z 772.338,A -85,B 0,C 180,E1 -17023.13,E2 -17023.13} C_VEL
LIN {X 0,Y 226.218,Z 768.472,A -85,B 0,C 180,E1 -17028.559,E2 -17028.559} C_VEL
LIN {X 0,Y 229.7,Z 762.535,A -85,B 0,C 180,E1 -17034.155,E2 -17034.155} C_VEL
LIN {X 0,Y 235.455,Z 754.321,A -85,B 0,C 180,E1 -17039.794,E2 -17039.794} C_VEL
LIN {X 0,Y 243.487,Z 744.149,A -85,B 0,C 180,E1 -17045.095,E2 -17045.095} C_VEL
LIN {X 0,Y 254.295,Z 731.59,A -85,B 0,C 180,E1 -17050.155,E2 -17050.155} C_VEL
LIN {X 0,Y 267.584,Z 717.288,A -85,B 0,C 180,E1 -17054.629,E2 -17054.629} C_VEL
LIN {X 0,Y 279.674,Z 705.089,A -85,B 0,C 180,E1 -17057.701,E2 -17057.701} C_VEL
LIN {X 0,Y 265.174,Z 717.754,A -85,B 0,C 180,E1 -17061.528,E2 -17061.528} C_VEL
LIN {X 0,Y 252.612,Z 729.11,A -85,B 0,C 180,E1 -17066.077,E2 -17066.077} C_VEL
LIN {X 0,Y 242.853,Z 738.169,A -85,B 0,C 180,E1 -17070.934,E2 -17070.934} C_VEL
LIN {X 0,Y 235.58,Z 744.978,A -85,B 0,C 180,E1 -17075.956,E2 -17075.956} C_VEL
LIN {X 0,Y 230.269,Z 749.837,A -85,B 0,C 180,E1 -17081.258,E2 -17081.258} C_VEL
LIN {X 0,Y 226.95,Z 752.62,A -85,B 0,C 180,E1 -17086.498,E2 -17086.498} C_VEL
LIN {X 0,Y 225.16,Z 753.534,A -85,B 0,C 180,E1 -17091.574,E2 -17091.574} C_VEL
LIN {X 0,Y 224.408,Z 752.743,A -85,B 0,C 180,E1 -17096.447,E2 -17096.447} C_VEL
LIN {X 0,Y 224.198,Z 750.439,A -85,B 0,C 180,E1 -17101.023,E2 -17101.023} C_VEL
LIN {X 0,Y 224.234,Z 746.715,A -85,B 0,C 180,E1 -17105.374,E2 -17105.374} C_VEL
LIN {X 0,Y 224.634,Z 741.414,A -85,B 0,C 180,E1 -17109.739,E2 -17109.739} C_VEL
LIN {X 0,Y 225.605,Z 734.39,A -85,B 0,C 180,E1 -17114.109,E2 -17114.109} C_VEL
LIN {X 0,Y 227.332,Z 725.447,A -85,B 0,C 180,E1 -17118.463,E2 -17118.463} C_VEL
LIN {X 0,Y 229.76,Z 715.051,A -85,B 0,C 180,E1 -17122.518,E2 -17122.518} C_VEL
LIN {X 0,Y 232.803,Z 703.296,A -85,B 0,C 180,E1 -17126.256,E2 -17126.256} C_VEL
LIN {X 0,Y 236.612,Z 689.242,A -85,B 0,C 180,E1 -17129.911,E2 -17129.911} C_VEL
LIN {X 0,Y 240.871,Z 673.589,A -85,B 0,C 180,E1 -17133.227,E2 -17133.227} C_VEL
LIN {X 0,Y 245.425,Z 656.201,A -85,B 0,C 180,E1 -17136.21,E2 -17136.21} C_VEL
LIN {X 0,Y 249.925,Z 637.749,A -85,B 0,C 180,E1 -17138.749,E2 -17138.749} C_VEL
LIN {X 0,Y 254.246,Z 618.089,A -85,B 0,C 180,E1 -17140.905,E2 -17140.905} C_VEL
LIN {X 0,Y 258.195,Z 597.49,A -85,B 0,C 180,E1 -17142.664,E2 -17142.664} C_VEL
LIN {X 0,Y 261.59,Z 576.13,A -85,B 0,C 180,E1 -17144.042,E2 -17144.042} C_VEL
LIN {X 0,Y 264.306,Z 553.841,A -85,B 0,C 180,E1 -17145.055,E2 -17145.055} C_VEL
LIN {X 0,Y 279.796,Z 408.146,A -85,B 0,C 180,E1 -17150.351,E2 -17150.351} C_VEL
LIN {X 0,Y 267.51,Z 384.104,A -85,B 0,C 180,E1 -17153.934,E2 -17153.934} C_VEL
LIN {X 0,Y 256.178,Z 363.663,A -85,B 0,C 180,E1 -17157.541,E2 -17157.541} C_VEL
LIN {X 0,Y 255.776,Z 362.628,A -85,B 0,C 180,E1 -17157.881,E2 -17157.881} C_VEL
LIN {X 0,Y 256.512,Z 364.958,A -85,B 0,C 180,E1 -17158.612,E2 -17158.612} C_VEL
LIN {X 0,Y 262.035,Z 379.972,A -85,B 0,C 180,E1 -17162.285,E2 -17162.285} C_VEL
LIN {X 0,Y 266.545,Z 394.897,A -85,B 0,C 180,E1 -17165.48,E2 -17165.48} C_VEL
LIN {X 0,Y 260.248,Z 437.782,A -85,B 0,C 180,E1 -17170.471,E2 -17170.471} C_VEL
LIN {X 0,Y 254.152,Z 480.628,A -85,B 0,C 180,E1 -17175.531,E2 -17175.531} C_VEL
LIN {X 0,Y 253.586,Z 486.33,A -85,B 0,C 180,E1 -17176.146,E2 -17176.146} C_VEL
LIN {X 0,Y 255.345,Z 513.166,A -85,B 0,C 180,E1 -17177.378,E2 -17177.378} C_VEL
LIN {X 0,Y 249.556,Z 630.626,A -85,B 0,C 180,E1 -17180.688,E2 -17180.688} C_VEL
LIN {X 0,Y 248.069,Z 646.977,A -85,B 0,C 180,E1 -17181.567,E2 -17181.567} C_VEL
LIN {X 0,Y 246.058,Z 662.048,A -85,B 0,C 180,E1 -17182.761,E2 -17182.761} C_VEL
LIN {X 0,Y 243.492,Z 676.649,A -85,B 0,C 180,E1 -17184.342,E2 -17184.342} C_VEL
LIN {X 0,Y 240.384,Z 691.194,A -85,B 0,C 180,E1 -17186.42,E2 -17186.42} C_VEL
LIN {X 0,Y 237.215,Z 703.971,A -85,B 0,C 180,E1 -17188.79,E2 -17188.79} C_VEL
LIN {X 0,Y 233.891,Z 716.252,A -85,B 0,C 180,E1 -17191.712,E2 -17191.712} C_VEL
LIN {X 0,Y 231.057,Z 726.056,A -85,B 0,C 180,E1 -17194.713,E2 -17194.713} C_VEL
LIN {X 0,Y 228.39,Z 735.262,A -85,B 0,C 180,E1 -17198.343,E2 -17198.343} C_VEL
LIN {X 0,Y 226.476,Z 742.158,A -85,B 0,C 180,E1 -17201.973,E2 -17201.973} C_VEL
LIN {X 0,Y 225.141,Z 747.679,A -85,B 0,C 180,E1 -17205.979,E2 -17205.979} C_VEL
LIN {X 0,Y 224.477,Z 751.264,A -85,B 0,C 180,E1 -17209.973,E2 -17209.973} C_VEL
LIN {X 0,Y 224.265,Z 753.211,A -85,B 0,C 180,E1 -17214.212,E2 -17214.212} C_VEL
LIN {X 0,Y 224.38,Z 753.375,A -85,B 0,C 180,E1 -17218.183,E2 -17218.183} C_VEL
LIN {X 0,Y 224.933,Z 751.769,A -85,B 0,C 180,E1 -17222.371,E2 -17222.371} C_VEL
LIN {X 0,Y 226.112,Z 748.514,A -85,B 0,C 180,E1 -17226.407,E2 -17226.407} C_VEL
LIN {X 0,Y 228.106,Z 743.271,A -85,B 0,C 180,E1 -17230.442,E2 -17230.442} C_VEL
LIN {X 0,Y 230.839,Z 736.383,A -85,B 0,C 180,E1 -17234.211,E2 -17234.211} C_VEL
LIN {X 0,Y 234.113,Z 727.94,A -85,B 0,C 180,E1 -17237.629,E2 -17237.629} C_VEL
LIN {X 0,Y 237.761,Z 718.16,A -85,B 0,C 180,E1 -17240.689,E2 -17240.689} C_VEL
LIN {X 0,Y 241.601,Z 706.878,A -85,B 0,C 180,E1 -17243.419,E2 -17243.419} C_VEL
LIN {X 0,Y 245.637,Z 693.669,A -85,B 0,C 180,E1 -17245.902,E2 -17245.902} C_VEL
LIN {X 0,Y 249.157,Z 680.091,A -85,B 0,C 180,E1 -17247.853,E2 -17247.853} C_VEL
LIN {X 0,Y 252.375,Z 665.07,A -85,B 0,C 180,E1 -17249.497,E2 -17249.497} C_VEL
LIN {X 0,Y 252.892,Z 658.091,A -85,B 0,C 180,E1 -17250.27,E2 -17250.27} C_VEL
LIN {X 0,Y 251.258,Z 644.385,A -85,B 0,C 180,E1 -17251.954,E2 -17251.954} C_VEL
LIN {X 0,Y 250.604,Z 636.11,A -85,B 0,C 180,E1 -17252.675,E2 -17252.675} C_VEL
LIN {X 0,Y 250.705,Z 632.868,A -85,B 0,C 180,E1 -17252.838,E2 -17252.838} C_VEL
LIN {X 0,Y 257.896,Z 513.32,A -85,B 0,C 180,E1 -17256.266,E2 -17256.266} C_VEL
LIN {X 0,Y 256.313,Z 487.239,A -85,B 0,C 180,E1 -17257.825,E2 -17257.825} C_VEL
LIN {X 0,Y 264.093,Z 441.625,A -85,B 0,C 180,E1 -17263.163,E2 -17263.163} C_VEL
LIN {X 0,Y 270.737,Z 404.278,A -85,B 0,C 180,E1 -17267.522,E2 -17267.522} C_VEL
LIN {X 0,Y 268.321,Z 393.587,A -85,B 0,C 180,E1 -17270.346,E2 -17270.346} C_VEL
LIN {X 0,Y 265.327,Z 384.015,A -85,B 0,C 180,E1 -17273.291,E2 -17273.291} C_VEL
LIN {X 0,Y 262.014,Z 374.57,A -85,B 0,C 180,E1 -17276.937,E2 -17276.937} C_VEL
LIN {X 0,Y 258.867,Z 366.992,A -85,B 0,C 180,E1 -17280.663,E2 -17280.663} C_VEL
LIN {X 0,Y 256.999,Z 362.781,A -85,B 0,C 180,E1 -17283.345,E2 -17283.345} C_VEL
LIN {X 0,Y 255.254,Z 358.691,A -85,B 0,C 180,E1 -17286.522,E2 -17286.522} C_VEL
LIN {X 0,Y 253.568,Z 354.666,A -85,B 0,C 180,E1 -17291.14,E2 -17291.14} C_VEL
LIN {X 0,Y 253.229,Z 353.955,A -85,B 0,C 180,E1 -17292.785,E2 -17292.785} C_VEL
LIN {X 0,Y 253.131,Z 353.618,A -85,B 0,C 180,E1 -17298.42,E2 -17298.42} C_VEL
LIN {X 0,Y 253.853,Z 354.345,A -85,B 0,C 180,E1 -17301.245,E2 -17301.245} C_VEL
LIN {X 0,Y 253.469,Z 359.89,A -85,B 0,C 180,E1 -17303.725,E2 -17303.725} C_VEL
LIN {X 0,Y 253.446,Z 366.618,A -85,B 0,C 180,E1 -17306.064,E2 -17306.064} C_VEL
LIN {X 0,Y 265.525,Z 387.341,A -85,B 0,C 180,E1 -17309.96,E2 -17309.96} C_VEL
LIN {X 0,Y 278.506,Z 411.075,A -85,B 0,C 180,E1 -17313.718,E2 -17313.718} C_VEL
LIN {X 0,Y 278.766,Z 412.273,A -85,B 0,C 180,E1 -17313.827,E2 -17313.827} C_VEL
LIN {X 0,Y 261.181,Z 575.534,A -85,B 0,C 180,E1 -17319.644,E2 -17319.644} C_VEL
LIN {X 0,Y 257.863,Z 597.286,A -85,B 0,C 180,E1 -17320.797,E2 -17320.797} C_VEL
LIN {X 0,Y 253.989,Z 617.808,A -85,B 0,C 180,E1 -17322.266,E2 -17322.266} C_VEL
LIN {X 0,Y 249.454,Z 638.208,A -85,B 0,C 180,E1 -17324.159,E2 -17324.159} C_VEL
LIN {X 0,Y 244.562,Z 657.679,A -85,B 0,C 180,E1 -17326.446,E2 -17326.446} C_VEL
LIN {X 0,Y 239.614,Z 675.697,A -85,B 0,C 180,E1 -17329.075,E2 -17329.075} C_VEL
LIN {X 0,Y 234.634,Z 692.797,A -85,B 0,C 180,E1 -17332.151,E2 -17332.151} C_VEL
LIN {X 0,Y 229.682,Z 709.307,A -85,B 0,C 180,E1 -17335.802,E2 -17335.802} C_VEL
LIN {X 0,Y 226.058,Z 725.598,A -85,B 0,C 180,E1 -17339.283,E2 -17339.283} C_VEL
LIN {X 0,Y 223.452,Z 736.747,A -85,B 0,C 180,E1 -17342.27,E2 -17342.27} C_VEL
LIN {X 0,Y 220.803,Z 747.635,A -85,B 0,C 180,E1 -17345.953,E2 -17345.953} C_VEL
LIN {X 0,Y 218.785,Z 756.288,A -85,B 0,C 180,E1 -17349.68,E2 -17349.68} C_VEL
LIN {X 0,Y 217.227,Z 763.841,A -85,B 0,C 180,E1 -17353.971,E2 -17353.971} C_VEL
LIN {X 0,Y 216.438,Z 769.056,A -85,B 0,C 180,E1 -17358.005,E2 -17358.005} C_VEL
LIN {X 0,Y 216.175,Z 772.697,A -85,B 0,C 180,E1 -17362.295,E2 -17362.295} C_VEL
LIN {X 0,Y 216.227,Z 774.497,A -85,B 0,C 180,E1 -17366.291,E2 -17366.291} C_VEL
LIN {X 0,Y 216.314,Z 774.74,A -85,B 0,C 180,E1 -17370.268,E2 -17370.268} C_VEL
LIN {X 0,Y 216.248,Z 774.064,A -85,B 0,C 180,E1 -17373.714,E2 -17373.714} C_VEL
LIN {X 0,Y 216.12,Z 773.83,A -85,B 0,C 180,E1 -17378.516,E2 -17378.516} C_VEL
LIN {X 0,Y 216.608,Z 772.136,A -85,B 0,C 180,E1 -17383.619,E2 -17383.619} C_VEL
LIN {X 0,Y 218.617,Z 768.29,A -85,B 0,C 180,E1 -17389.507,E2 -17389.507} C_VEL
LIN {X 0,Y 222.507,Z 762.588,A -85,B 0,C 180,E1 -17395.273,E2 -17395.273} C_VEL
LIN {X 0,Y 228.901,Z 754.64,A -85,B 0,C 180,E1 -17401.115,E2 -17401.115} C_VEL
LIN {X 0,Y 237.898,Z 744.644,A -85,B 0,C 180,E1 -17406.645,E2 -17406.645} C_VEL
LIN {X 0,Y 249.536,Z 732.752,A -85,B 0,C 180,E1 -17411.696,E2 -17411.696} C_VEL
LIN {X 0,Y 264.301,Z 718.748,A -85,B 0,C 180,E1 -17416.269,E2 -17416.269} C_VEL
LIN {X 0,Y 270.243,Z 713.321,A -85,B 0,C 180,E1 -17417.731,E2 -17417.731} C_VEL
LIN {X 0,Y 254.966,Z 725.279,A -85,B 0,C 180,E1 -17421.999,E2 -17421.999} C_VEL
LIN {X 0,Y 242.522,Z 735.299,A -85,B 0,C 180,E1 -17426.82,E2 -17426.82} C_VEL
LIN {X 0,Y 233.128,Z 742.927,A -85,B 0,C 180,E1 -17431.851,E2 -17431.851} C_VEL
LIN {X 0,Y 226.145,Z 748.507,A -85,B 0,C 180,E1 -17437.104,E2 -17437.104} C_VEL
LIN {X 0,Y 221.197,Z 752.221,A -85,B 0,C 180,E1 -17442.643,E2 -17442.643} C_VEL
LIN {X 0,Y 218.355,Z 753.923,A -85,B 0,C 180,E1 -17447.841,E2 -17447.841} C_VEL
LIN {X 0,Y 216.847,Z 753.922,A -85,B 0,C 180,E1 -17453.116,E2 -17453.116} C_VEL
LIN {X 0,Y 216.309,Z 752.398,A -85,B 0,C 180,E1 -17457.882,E2 -17457.882} C_VEL
LIN {X 0,Y 216.179,Z 749.422,A -85,B 0,C 180,E1 -17462.473,E2 -17462.473} C_VEL
LIN {X 0,Y 216.321,Z 745.098,A -85,B 0,C 180,E1 -17466.903,E2 -17466.903} C_VEL
LIN {X 0,Y 216.981,Z 738.666,A -85,B 0,C 180,E1 -17471.699,E2 -17471.699} C_VEL
LIN {X 0,Y 218.301,Z 730.723,A -85,B 0,C 180,E1 -17476.225,E2 -17476.225} C_VEL
LIN {X 0,Y 220.483,Z 720.753,A -85,B 0,C 180,E1 -17480.716,E2 -17480.716} C_VEL
LIN {X 0,Y 223.414,Z 709.249,A -85,B 0,C 180,E1 -17484.879,E2 -17484.879} C_VEL
LIN {X 0,Y 227.1,Z 695.837,A -85,B 0,C 180,E1 -17488.815,E2 -17488.815} C_VEL
LIN {X 0,Y 231.34,Z 680.776,A -85,B 0,C 180,E1 -17492.408,E2 -17492.408} C_VEL
LIN {X 0,Y 235.948,Z 664.01,A -85,B 0,C 180,E1 -17495.64,E2 -17495.64} C_VEL
LIN {X 0,Y 240.593,Z 646.172,A -85,B 0,C 180,E1 -17498.412,E2 -17498.412} C_VEL
LIN {X 0,Y 245.292,Z 626.405,A -85,B 0,C 180,E1 -17500.863,E2 -17500.863} C_VEL
LIN {X 0,Y 249.469,Z 606.611,A -85,B 0,C 180,E1 -17502.794,E2 -17502.794} C_VEL
LIN {X 0,Y 253.18,Z 585.962,A -85,B 0,C 180,E1 -17504.349,E2 -17504.349} C_VEL
LIN {X 0,Y 256.316,Z 564.259,A -85,B 0,C 180,E1 -17505.541,E2 -17505.541} C_VEL
LIN {X 0,Y 273.266,Z 410.887,A -85,B 0,C 180,E1 -17511.333,E2 -17511.333} C_VEL
LIN {X 0,Y 262.067,Z 388.774,A -85,B 0,C 180,E1 -17514.72,E2 -17514.72} C_VEL
LIN {X 0,Y 252.395,Z 371.07,A -85,B 0,C 180,E1 -17517.902,E2 -17517.902} C_VEL
LIN {X 0,Y 251.628,Z 371.456,A -85,B 0,C 180,E1 -17518.326,E2 -17518.326} C_VEL
LIN {X 0,Y 256.638,Z 386.082,A -85,B 0,C 180,E1 -17521.998,E2 -17521.998} C_VEL
LIN {X 0,Y 260.149,Z 397.891,A -85,B 0,C 180,E1 -17524.584,E2 -17524.584} C_VEL
LIN {X 0,Y 253.926,Z 438.358,A -85,B 0,C 180,E1 -17529.363,E2 -17529.363} C_VEL
LIN {X 0,Y 247.536,Z 481.768,A -85,B 0,C 180,E1 -17534.536,E2 -17534.536} C_VEL
LIN {X 0,Y 247.05,Z 486.725,A -85,B 0,C 180,E1 -17535.068,E2 -17535.068} C_VEL
LIN {X 0,Y 248.738,Z 513.972,A -85,B 0,C 180,E1 -17536.36,E2 -17536.36} C_VEL
LIN {X 0,Y 242.7,Z 631.12,A -85,B 0,C 180,E1 -17539.734,E2 -17539.734} C_VEL
LIN {X 0,Y 241.14,Z 647.499,A -85,B 0,C 180,E1 -17540.637,E2 -17540.637} C_VEL
LIN {X 0,Y 238.914,Z 663.402,A -85,B 0,C 180,E1 -17541.938,E2 -17541.938} C_VEL
LIN {X 0,Y 236.059,Z 678.632,A -85,B 0,C 180,E1 -17543.675,E2 -17543.675} C_VEL
LIN {X 0,Y 232.846,Z 692.861,A -85,B 0,C 180,E1 -17545.811,E2 -17545.811} C_VEL
LIN {X 0,Y 229.366,Z 706.104,A -85,B 0,C 180,E1 -17548.412,E2 -17548.412} C_VEL
LIN {X 0,Y 226.131,Z 717.449,A -85,B 0,C 180,E1 -17551.264,E2 -17551.264} C_VEL
LIN {X 0,Y 222.981,Z 727.817,A -85,B 0,C 180,E1 -17554.627,E2 -17554.627} C_VEL
LIN {X 0,Y 220.478,Z 736.081,A -85,B 0,C 180,E1 -17558.079,E2 -17558.079} C_VEL
LIN {X 0,Y 218.37,Z 743.358,A -85,B 0,C 180,E1 -17562.156,E2 -17562.156} C_VEL
LIN {X 0,Y 217.125,Z 748.36,A -85,B 0,C 180,E1 -17566.036,E2 -17566.036} C_VEL
LIN {X 0,Y 216.449,Z 751.904,A -85,B 0,C 180,E1 -17570.323,E2 -17570.323} C_VEL
LIN {X 0,Y 216.272,Z 753.681,A -85,B 0,C 180,E1 -17574.584,E2 -17574.584} C_VEL
LIN {X 0,Y 216.431,Z 753.708,A -85,B 0,C 180,E1 -17578.711,E2 -17578.711} C_VEL
LIN {X 0,Y 217.129,Z 751.913,A -85,B 0,C 180,E1 -17583.225,E2 -17583.225} C_VEL
LIN {X 0,Y 218.538,Z 748.345,A -85,B 0,C 180,E1 -17587.477,E2 -17587.477} C_VEL
LIN {X 0,Y 220.87,Z 742.794,A -85,B 0,C 180,E1 -17591.713,E2 -17591.713} C_VEL
LIN {X 0,Y 223.81,Z 735.833,A -85,B 0,C 180,E1 -17595.46,E2 -17595.46} C_VEL
LIN {X 0,Y 227.565,Z 726.772,A -85,B 0,C 180,E1 -17599.104,E2 -17599.104} C_VEL
LIN {X 0,Y 231.512,Z 716.57,A -85,B 0,C 180,E1 -17602.212,E2 -17602.212} C_VEL
LIN {X 0,Y 235.837,Z 704.394,A -85,B 0,C 180,E1 -17605.085,E2 -17605.085} C_VEL
LIN {X 0,Y 239.957,Z 691.059,A -85,B 0,C 180,E1 -17607.484,E2 -17607.484} C_VEL
LIN {X 0,Y 243.641,Z 677.153,A -85,B 0,C 180,E1 -17609.41,E2 -17609.41} C_VEL
LIN {X 0,Y 246.771,Z 662.268,A -85,B 0,C 180,E1 -17610.95,E2 -17610.95} C_VEL
LIN {X 0,Y 249.311,Z 646.144,A -85,B 0,C 180,E1 -17612.16,E2 -17612.16} C_VEL
LIN {X 0,Y 250.705,Z 632.868,A -85,B 0,C 180,E1 -17612.838,E2 -17612.838} C_VEL
LIN {X 0,Y 250.506,Z 625.322,A -85,B 0,C 180,E1 -17613.262,E2 -17613.262} C_VEL
LIN {X 0,Y 247.179,Z 605.498,A -85,B 0,C 180,E1 -17614.839,E2 -17614.839} C_VEL
LIN {X 0,Y 247.044,Z 598.979,A -85,B 0,C 180,E1 -17615.143,E2 -17615.143} C_VEL
LIN {X 0,Y 252.379,Z 514.396,A -85,B 0,C 180,E1 -17617.553,E2 -17617.553} C_VEL
LIN {X 0,Y 250.911,Z 487.444,A -85,B 0,C 180,E1 -17619.227,E2 -17619.227} C_VEL
LIN {X 0,Y 258.854,Z 443.464,A -85,B 0,C 180,E1 -17624.427,E2 -17624.427} C_VEL
LIN {X 0,Y 265.455,Z 408.125,A -85,B 0,C 180,E1 -17628.594,E2 -17628.594} C_VEL
LIN {X 0,Y 263.242,Z 397.681,A -85,B 0,C 180,E1 -17631.48,E2 -17631.48} C_VEL
LIN {X 0,Y 260.693,Z 389.136,A -85,B 0,C 180,E1 -17634.276,E2 -17634.276} C_VEL
LIN {X 0,Y 257.967,Z 380.891,A -85,B 0,C 180,E1 -17637.556,E2 -17637.556} C_VEL
LIN {X 0,Y 255.306,Z 373.868,A -85,B 0,C 180,E1 -17641.121,E2 -17641.121} C_VEL
LIN {X 0,Y 253.468,Z 369.676,A -85,B 0,C 180,E1 -17643.844,E2 -17643.844} C_VEL
LIN {X 0,Y 252.046,Z 365.92,A -85,B 0,C 180,E1 -17646.834,E2 -17646.834} C_VEL
LIN {X 0,Y 250.652,Z 361.942,A -85,B 0,C 180,E1 -17651.504,E2 -17651.504} C_VEL
LIN {X 0,Y 250.057,Z 361.041,A -85,B 0,C 180,E1 -17655.777,E2 -17655.777} C_VEL
LIN {X 0,Y 251.049,Z 361.654,A -85,B 0,C 180,E1 -17660.76,E2 -17660.76} C_VEL
LIN {X 0,Y 250.59,Z 366.24,A -85,B 0,C 180,E1 -17662.833,E2 -17662.833} C_VEL
LIN {X 0,Y 250.315,Z 374.957,A -85,B 0,C 180,E1 -17665.905,E2 -17665.905} C_VEL
LIN {X 0,Y 262.393,Z 396.063,A -85,B 0,C 180,E1 -17669.851,E2 -17669.851} C_VEL
LIN {X 0,Y 272.396,Z 414.775,A -85,B 0,C 180,E1 -17672.829,E2 -17672.829} C_VEL
LIN {X 0,Y 254.432,Z 575.008,A -85,B 0,C 180,E1 -17678.69,E2 -17678.69} C_VEL
LIN {X 0,Y 251.039,Z 596.637,A -85,B 0,C 180,E1 -17679.859,E2 -17679.859} C_VEL
LIN {X 0,Y 246.795,Z 618.373,A -85,B 0,C 180,E1 -17681.457,E2 -17681.457} C_VEL
LIN {X 0,Y 242.147,Z 638.593,A -85,B 0,C 180,E1 -17683.392,E2 -17683.392} C_VEL
LIN {X 0,Y 237.085,Z 658.088,A -85,B 0,C 180,E1 -17685.757,E2 -17685.757} C_VEL
LIN {X 0,Y 231.842,Z 676.526,A -85,B 0,C 180,E1 -17688.552,E2 -17688.552} C_VEL
LIN {X 0,Y 226.791,Z 693.347,A -85,B 0,C 180,E1 -17691.697,E2 -17691.697} C_VEL
LIN {X 0,Y 224.95,Z 699.747,A -85,B 0,C 180,E1 -17692.971,E2 -17692.971} C_VEL
LIN {X 0,Y 222.22,Z 712.919,A -85,B 0,C 180,E1 -17695.311,E2 -17695.311} C_VEL
LIN {X 0,Y 219.129,Z 725.901,A -85,B 0,C 180,E1 -17698.2,E2 -17698.2} C_VEL
LIN {X 0,Y 216.268,Z 736.876,A -85,B 0,C 180,E1 -17701.265,E2 -17701.265} C_VEL
LIN {X 0,Y 213.368,Z 747.654,A -85,B 0,C 180,E1 -17705.059,E2 -17705.059} C_VEL
LIN {X 0,Y 211.132,Z 756.177,A -85,B 0,C 180,E1 -17708.909,E2 -17708.909} C_VEL
LIN {X 0,Y 209.394,Z 763.67,A -85,B 0,C 180,E1 -17713.355,E2 -17713.355} C_VEL
LIN {X 0,Y 208.494,Z 768.795,A -85,B 0,C 180,E1 -17717.541,E2 -17717.541} C_VEL
LIN {X 0,Y 208.185,Z 772.382,A -85,B 0,C 180,E1 -17721.997,E2 -17721.997} C_VEL
LIN {X 0,Y 208.229,Z 774.139,A -85,B 0,C 180,E1 -17726.148,E2 -17726.148} C_VEL
LIN {X 0,Y 208.33,Z 774.357,A -85,B 0,C 180,E1 -17730.003,E2 -17730.003} C_VEL
LIN {X 0,Y 208.255,Z 773.413,A -85,B 0,C 180,E1 -17734.133,E2 -17734.133} C_VEL
LIN {X 0,Y 208.138,Z 773.329,A -85,B 0,C 180,E1 -17739.124,E2 -17739.124} C_VEL
LIN {X 0,Y 208.839,Z 771.599,A -85,B 0,C 180,E1 -17744.737,E2 -17744.737} C_VEL
LIN {X 0,Y 211.226,Z 767.895,A -85,B 0,C 180,E1 -17750.797,E2 -17750.797} C_VEL
LIN {X 0,Y 215.656,Z 762.405,A -85,B 0,C 180,E1 -17756.729,E2 -17756.729} C_VEL
LIN {X 0,Y 222.999,Z 754.531,A -85,B 0,C 180,E1 -17762.859,E2 -17762.859} C_VEL
LIN {X 0,Y 233.47,Z 744.408,A -85,B 0,C 180,E1 -17768.704,E2 -17768.704} C_VEL
LIN {X 0,Y 246.738,Z 732.553,A -85,B 0,C 180,E1 -17773.866,E2 -17773.866} C_VEL
LIN {X 0,Y 260.577,Z 720.951,A -85,B 0,C 180,E1 -17777.819,E2 -17777.819} C_VEL
LIN {X 0,Y 245.831,Z 731.225,A -85,B 0,C 180,E1 -17782.11,E2 -17782.11} C_VEL
LIN {X 0,Y 233.535,Z 739.915,A -85,B 0,C 180,E1 -17787.062,E2 -17787.062} C_VEL
LIN {X 0,Y 223.739,Z 746.776,A -85,B 0,C 180,E1 -17792.595,E2 -17792.595} C_VEL
LIN {X 0,Y 216.732,Z 751.437,A -85,B 0,C 180,E1 -17798.343,E2 -17798.343} C_VEL
LIN {X 0,Y 212.347,Z 753.972,A -85,B 0,C 180,E1 -17803.872,E2 -17803.872} C_VEL
LIN {X 0,Y 209.814,Z 754.763,A -85,B 0,C 180,E1 -17809.29,E2 -17809.29} C_VEL
LIN {X 0,Y 208.627,Z 753.948,A -85,B 0,C 180,E1 -17814.501,E2 -17814.501} C_VEL
LIN {X 0,Y 208.24,Z 751.631,A -85,B 0,C 180,E1 -17819.451,E2 -17819.451} C_VEL
LIN {X 0,Y 208.192,Z 747.984,A -85,B 0,C 180,E1 -17824.132,E2 -17824.132} C_VEL
LIN {X 0,Y 208.52,Z 742.631,A -85,B 0,C 180,E1 -17828.954,E2 -17828.954} C_VEL
LIN {X 0,Y 209.469,Z 735.428,A -85,B 0,C 180,E1 -17833.809,E2 -17833.809} C_VEL
LIN {X 0,Y 211.218,Z 726.507,A -85,B 0,C 180,E1 -17838.493,E2 -17838.493} C_VEL
LIN {X 0,Y 213.734,Z 716.142,A -85,B 0,C 180,E1 -17842.849,E2 -17842.849} C_VEL
LIN {X 0,Y 217.162,Z 703.568,A -85,B 0,C 180,E1 -17847.119,E2 -17847.119} C_VEL
LIN {X 0,Y 221.23,Z 689.419,A -85,B 0,C 180,E1 -17851.014,E2 -17851.014} C_VEL
LIN {X 0,Y 225.803,Z 673.604,A -85,B 0,C 180,E1 -17854.548,E2 -17854.548} C_VEL
LIN {X 0,Y 230.439,Z 656.926,A -85,B 0,C 180,E1 -17857.563,E2 -17857.563} C_VEL
LIN {X 0,Y 235.234,Z 638.439,A -85,B 0,C 180,E1 -17860.248,E2 -17860.248} C_VEL
LIN {X 0,Y 239.786,Z 619.029,A -85,B 0,C 180,E1 -17862.495,E2 -17862.495} C_VEL
LIN {X 0,Y 244.082,Z 598.091,A -85,B 0,C 180,E1 -17864.385,E2 -17864.385} C_VEL
LIN {X 0,Y 247.764,Z 576.507,A -85,B 0,C 180,E1 -17865.855,E2 -17865.855} C_VEL
LIN {X 0,Y 250.673,Z 554.428,A -85,B 0,C 180,E1 -17866.917,E2 -17866.917} C_VEL
LIN {X 0,Y 266.856,Z 413.714,A -85,B 0,C 180,E1 -17872.325,E2 -17872.325} C_VEL
LIN {X 0,Y 255.082,Z 390.415,A -85,B 0,C 180,E1 -17876.041,E2 -17876.041} C_VEL
LIN {X 0,Y 249.203,Z 379.769,A -85,B 0,C 180,E1 -17878.018,E2 -17878.018} C_VEL
LIN {X 0,Y 247.528,Z 379.986,A -85,B 0,C 180,E1 -17878.543,E2 -17878.543} C_VEL
LIN {X 0,Y 247.772,Z 381.516,A -85,B 0,C 180,E1 -17879.064,E2 -17879.064} C_VEL
LIN {X 0,Y 252.534,Z 396.462,A -85,B 0,C 180,E1 -17882.657,E2 -17882.657} C_VEL
LIN {X 0,Y 253.805,Z 401.186,A -85,B 0,C 180,E1 -17883.69,E2 -17883.69} C_VEL
LIN {X 0,Y 247.15,Z 442.761,A -85,B 0,C 180,E1 -17888.645,E2 -17888.645} C_VEL
LIN {X 0,Y 240.542,Z 486.564,A -85,B 0,C 180,E1 -17893.912,E2 -17893.912} C_VEL
LIN {X 0,Y 242.209,Z 514.736,A -85,B 0,C 180,E1 -17895.287,E2 -17895.287} C_VEL
LIN {X 0,Y 235.918,Z 631.475,A -85,B 0,C 180,E1 -17898.721,E2 -17898.721} C_VEL
LIN {X 0,Y 234.284,Z 647.929,A -85,B 0,C 180,E1 -17899.648,E2 -17899.648} C_VEL
LIN {X 0,Y 232.019,Z 663.507,A -85,B 0,C 180,E1 -17900.948,E2 -17900.948} C_VEL
LIN {X 0,Y 229.18,Z 678.184,A -85,B 0,C 180,E1 -17902.64,E2 -17902.64} C_VEL
LIN {X 0,Y 225.917,Z 692.2,A -85,B 0,C 180,E1 -17904.759,E2 -17904.759} C_VEL
LIN {X 0,Y 222.426,Z 705.074,A -85,B 0,C 180,E1 -17907.292,E2 -17907.292} C_VEL
LIN {X 0,Y 218.942,Z 716.84,A -85,B 0,C 180,E1 -17910.259,E2 -17910.259} C_VEL
LIN {X 0,Y 215.822,Z 726.693,A -85,B 0,C 180,E1 -17913.45,E2 -17913.45} C_VEL
LIN {X 0,Y 212.897,Z 735.839,A -85,B 0,C 180,E1 -17917.282,E2 -17917.282} C_VEL
LIN {X 0,Y 210.739,Z 742.863,A -85,B 0,C 180,E1 -17921.214,E2 -17921.214} C_VEL
LIN {X 0,Y 209.246,Z 748.409,A -85,B 0,C 180,E1 -17925.518,E2 -17925.518} C_VEL
LIN {X 0,Y 208.528,Z 751.898,A -85,B 0,C 180,E1 -17929.608,E2 -17929.608} C_VEL
LIN {X 0,Y 208.282,Z 753.907,A -85,B 0,C 180,E1 -17934.078,E2 -17934.078} C_VEL
LIN {X 0,Y 208.413,Z 754.218,A -85,B 0,C 180,E1 -17938.352,E2 -17938.352} C_VEL
LIN {X 0,Y 209.021,Z 752.836,A -85,B 0,C 180,E1 -17942.716,E2 -17942.716} C_VEL
LIN {X 0,Y 210.373,Z 749.7,A -85,B 0,C 180,E1 -17947.124,E2 -17947.124} C_VEL
LIN {X 0,Y 212.475,Z 745.045,A -85,B 0,C 180,E1 -17951.204,E2 -17951.204} C_VEL
LIN {X 0,Y 215.469,Z 738.451,A -85,B 0,C 180,E1 -17955.228,E2 -17955.228} C_VEL
LIN {X 0,Y 219.129,Z 730.303,A -85,B 0,C 180,E1 -17958.923,E2 -17958.923} C_VEL
LIN {X 0,Y 223.412,Z 720.13,A -85,B 0,C 180,E1 -17962.381,E2 -17962.381} C_VEL
LIN {X 0,Y 227.614,Z 709.314,A -85,B 0,C 180,E1 -17965.224,E2 -17965.224} C_VEL
LIN {X 0,Y 232.077,Z 696.286,A -85,B 0,C 180,E1 -17967.849,E2 -17967.849} C_VEL
LIN {X 0,Y 235.875,Z 683.505,A -85,B 0,C 180,E1 -17969.847,E2 -17969.847} C_VEL
LIN {X 0,Y 239.41,Z 669.015,A -85,B 0,C 180,E1 -17971.568,E2 -17971.568} C_VEL
LIN {X 0,Y 242.243,Z 654.165,A -85,B 0,C 180,E1 -17972.885,E2 -17972.885} C_VEL
LIN {X 0,Y 244.365,Z 638.259,A -85,B 0,C 180,E1 -17973.864,E2 -17973.864} C_VEL
LIN {X 0,Y 245.77,Z 619.713,A -85,B 0,C 180,E1 -17974.55,E2 -17974.55} C_VEL
LIN {X 0,Y 247.044,Z 598.979,A -85,B 0,C 180,E1 -17975.143,E2 -17975.143} C_VEL
LIN {X 0,Y 246.824,Z 591.391,A -85,B 0,C 180,E1 -17975.524,E2 -17975.524} C_VEL
LIN {X 0,Y 243.808,Z 571.542,A -85,B 0,C 180,E1 -17977.151,E2 -17977.151} C_VEL
LIN {X 0,Y 243.739,Z 565.021,A -85,B 0,C 180,E1 -17977.467,E2 -17977.467} C_VEL
LIN {X 0,Y 247.01,Z 515.369,A -85,B 0,C 180,E1 -17978.906,E2 -17978.906} C_VEL
LIN {X 0,Y 245.652,Z 488.238,A -85,B 0,C 180,E1 -17980.638,E2 -17980.638} C_VEL
LIN {X 0,Y 254.225,Z 443.085,A -85,B 0,C 180,E1 -17986.013,E2 -17986.013} C_VEL
LIN {X 0,Y 260.412,Z 412.111,A -85,B 0,C 180,E1 -17989.715,E2 -17989.715} C_VEL
LIN {X 0,Y 258.365,Z 402.518,A -85,B 0,C 180,E1 -17992.438,E2 -17992.438} C_VEL
LIN {X 0,Y 256.136,Z 393.747,A -85,B 0,C 180,E1 -17995.521,E2 -17995.521} C_VEL
LIN {X 0,Y 253.566,Z 386.286,A -85,B 0,C 180,E1 -17998.643,E2 -17998.643} C_VEL
LIN {X 0,Y 251.427,Z 380.065,A -85,B 0,C 180,E1 -18002.05,E2 -18002.05} C_VEL
LIN {X 0,Y 250.014,Z 376.591,A -85,B 0,C 180,E1 -18004.357,E2 -18004.357} C_VEL
LIN {X 0,Y 248.907,Z 373.157,A -85,B 0,C 180,E1 -18007.188,E2 -18007.188} C_VEL
LIN {X 0,Y 247.67,Z 369.022,A -85,B 0,C 180,E1 -18012.354,E2 -18012.354} C_VEL
LIN {X 0,Y 247.621,Z 368.632,A -85,B 0,C 180,E1 -18018.114,E2 -18018.114} C_VEL
LIN {X 0,Y 248.197,Z 369.164,A -85,B 0,C 180,E1 -18020.393,E2 -18020.393} C_VEL
LIN {X 0,Y 247.706,Z 372.966,A -85,B 0,C 180,E1 -18022.048,E2 -18022.048} C_VEL
LIN {X 0,Y 247.234,Z 383.401,A -85,B 0,C 180,E1 -18025.768,E2 -18025.768} C_VEL
LIN {X 0,Y 260.302,Z 406.834,A -85,B 0,C 180,E1 -18030.083,E2 -18030.083} C_VEL
LIN {X 0,Y 265.966,Z 417.879,A -85,B 0,C 180,E1 -18031.823,E2 -18031.823} C_VEL
LIN {X 0,Y 247.654,Z 574.88,A -85,B 0,C 180,E1 -18037.72,E2 -18037.72} C_VEL
LIN {X 0,Y 244.008,Z 597.232,A -85,B 0,C 180,E1 -18038.97,E2 -18038.97} C_VEL
LIN {X 0,Y 239.656,Z 618.703,A -85,B 0,C 180,E1 -18040.601,E2 -18040.601} C_VEL
LIN {X 0,Y 234.816,Z 639.044,A -85,B 0,C 180,E1 -18042.611,E2 -18042.611} C_VEL
LIN {X 0,Y 229.483,Z 658.904,A -85,B 0,C 180,E1 -18045.107,E2 -18045.107} C_VEL
LIN {X 0,Y 223.881,Z 677.931,A -85,B 0,C 180,E1 -18048.117,E2 -18048.117} C_VEL
LIN {X 0,Y 221.404,Z 686.158,A -85,B 0,C 180,E1 -18049.61,E2 -18049.61} C_VEL
LIN {X 0,Y 218.973,Z 698.995,A -85,B 0,C 180,E1 -18051.449,E2 -18051.449} C_VEL
LIN {X 0,Y 215.945,Z 712.149,A -85,B 0,C 180,E1 -18053.823,E2 -18053.823} C_VEL
LIN {X 0,Y 212.554,Z 725.18,A -85,B 0,C 180,E1 -18056.773,E2 -18056.773} C_VEL
LIN {X 0,Y 209.385,Z 736.197,A -85,B 0,C 180,E1 -18059.911,E2 -18059.911} C_VEL
LIN {X 0,Y 206.173,Z 746.992,A -85,B 0,C 180,E1 -18063.816,E2 -18063.816} C_VEL
LIN {X 0,Y 203.671,Z 755.576,A -85,B 0,C 180,E1 -18067.793,E2 -18067.793} C_VEL
LIN {X 0,Y 201.684,Z 763.092,A -85,B 0,C 180,E1 -18072.401,E2 -18072.401} C_VEL
LIN {X 0,Y 200.61,Z 768.274,A -85,B 0,C 180,E1 -18076.749,E2 -18076.749} C_VEL
LIN {X 0,Y 200.197,Z 771.94,A -85,B 0,C 180,E1 -18081.445,E2 -18081.445} C_VEL
LIN {X 0,Y 200.221,Z 773.706,A -85,B 0,C 180,E1 -18085.707,E2 -18085.707} C_VEL
LIN {X 0,Y 200.333,Z 773.971,A -85,B 0,C 180,E1 -18089.717,E2 -18089.717} C_VEL
LIN {X 0,Y 200.295,Z 772.826,A -85,B 0,C 180,E1 -18093.724,E2 -18093.724} C_VEL
LIN {X 0,Y 200.16,Z 772.82,A -85,B 0,C 180,E1 -18099.491,E2 -18099.491} C_VEL
LIN {X 0,Y 200.96,Z 771.316,A -85,B 0,C 180,E1 -18105.293,E2 -18105.293} C_VEL
LIN {X 0,Y 203.772,Z 767.741,A -85,B 0,C 180,E1 -18111.898,E2 -18111.898} C_VEL
LIN {X 0,Y 209.25,Z 762.034,A -85,B 0,C 180,E1 -18118.547,E2 -18118.547} C_VEL
LIN {X 0,Y 217.872,Z 754.105,A -85,B 0,C 180,E1 -18125.008,E2 -18125.008} C_VEL
LIN {X 0,Y 229.955,Z 743.969,A -85,B 0,C 180,E1 -18131.041,E2 -18131.041} C_VEL
LIN {X 0,Y 245.059,Z 732.211,A -85,B 0,C 180,E1 -18136.237,E2 -18136.237} C_VEL
LIN {X 0,Y 250.94,Z 727.824,A -85,B 0,C 180,E1 -18137.864,E2 -18137.864} C_VEL
LIN {X 0,Y 236.066,Z 736.975,A -85,B 0,C 180,E1 -18142.418,E2 -18142.418} C_VEL
LIN {X 0,Y 223.912,Z 744.431,A -85,B 0,C 180,E1 -18147.599,E2 -18147.599} C_VEL
LIN {X 0,Y 214.325,Z 750.091,A -85,B 0,C 180,E1 -18153.395,E2 -18153.395} C_VEL
LIN {X 0,Y 207.845,Z 753.565,A -85,B 0,C 180,E1 -18159.147,E2 -18159.147} C_VEL
LIN {X 0,Y 203.692,Z 755.226,A -85,B 0,C 180,E1 -18164.921,E2 -18164.921} C_VEL
LIN {X 0,Y 201.414,Z 755.191,A -85,B 0,C 180,E1 -18170.572,E2 -18170.572} C_VEL
LIN {X 0,Y 200.441,Z 753.513,A -85,B 0,C 180,E1 -18176.111,E2 -18176.111} C_VEL
LIN {X 0,Y 200.194,Z 750.466,A -85,B 0,C 180,E1 -18181.146,E2 -18181.146} C_VEL
LIN {X 0,Y 200.265,Z 746.046,A -85,B 0,C 180,E1 -18186.019,E2 -18186.019} C_VEL
LIN {X 0,Y 200.8,Z 740.01,A -85,B 0,C 180,E1 -18190.908,E2 -18190.908} C_VEL
LIN {X 0,Y 202.065,Z 732.181,A -85,B 0,C 180,E1 -18195.793,E2 -18195.793} C_VEL
LIN {X 0,Y 204.249,Z 722.337,A -85,B 0,C 180,E1 -18200.639,E2 -18200.639} C_VEL
LIN {X 0,Y 207.251,Z 710.975,A -85,B 0,C 180,E1 -18205.123,E2 -18205.123} C_VEL
LIN {X 0,Y 211.07,Z 697.754,A -85,B 0,C 180,E1 -18209.347,E2 -18209.347} C_VEL
LIN {X 0,Y 215.499,Z 682.9,A -85,B 0,C 180,E1 -18213.196,E2 -18213.196} C_VEL
LIN {X 0,Y 220.332,Z 666.479,A -85,B 0,C 180,E1 -18216.638,E2 -18216.638} C_VEL
LIN {X 0,Y 225.199,Z 649.082,A -85,B 0,C 180,E1 -18219.579,E2 -18219.579} C_VEL
LIN {X 0,Y 230.125,Z 629.881,A -85,B 0,C 180,E1 -18222.167,E2 -18222.167} C_VEL
LIN {X 0,Y 234.746,Z 609.704,A -85,B 0,C 180,E1 -18224.31,E2 -18224.31} C_VEL
LIN {X 0,Y 238.893,Z 588.471,A -85,B 0,C 180,E1 -18226.047,E2 -18226.047} C_VEL
LIN {X 0,Y 242.386,Z 566.631,A -85,B 0,C 180,E1 -18227.356,E2 -18227.356} C_VEL
LIN {X 0,Y 260.37,Z 416.349,A -85,B 0,C 180,E1 -18233.366,E2 -18233.366} C_VEL
LIN {X 0,Y 249.217,Z 394.288,A -85,B 0,C 180,E1 -18237.033,E2 -18237.033} C_VEL
LIN {X 0,Y 246.051,Z 388.346,A -85,B 0,C 180,E1 -18238.137,E2 -18238.137} C_VEL
LIN {X 0,Y 243.328,Z 388.829,A -85,B 0,C 180,E1 -18238.851,E2 -18238.851} C_VEL
LIN {X 0,Y 243.265,Z 389.649,A -85,B 0,C 180,E1 -18239.209,E2 -18239.209} C_VEL
LIN {X 0,Y 247.504,Z 404.236,A -85,B 0,C 180,E1 -18242.719,E2 -18242.719} C_VEL
LIN {X 0,Y 240.851,Z 444.3,A -85,B 0,C 180,E1 -18247.545,E2 -18247.545} C_VEL
LIN {X 0,Y 234.151,Z 487.041,A -85,B 0,C 180,E1 -18252.733,E2 -18252.733} C_VEL
LIN {X 0,Y 235.723,Z 515.556,A -85,B 0,C 180,E1 -18254.171,E2 -18254.171} C_VEL
LIN {X 0,Y 229.181,Z 631.841,A -85,B 0,C 180,E1 -18257.662,E2 -18257.662} C_VEL
LIN {X 0,Y 227.486,Z 648.235,A -85,B 0,C 180,E1 -18258.604,E2 -18258.604} C_VEL
LIN {X 0,Y 225.189,Z 663.46,A -85,B 0,C 180,E1 -18259.896,E2 -18259.896} C_VEL
LIN {X 0,Y 222.291,Z 677.993,A -85,B 0,C 180,E1 -18261.591,E2 -18261.591} C_VEL
LIN {X 0,Y 218.776,Z 692.523,A -85,B 0,C 180,E1 -18263.832,E2 -18263.832} C_VEL
LIN {X 0,Y 215.175,Z 705.27,A -85,B 0,C 180,E1 -18266.401,E2 -18266.401} C_VEL
LIN {X 0,Y 211.522,Z 717.075,A -85,B 0,C 180,E1 -18269.455,E2 -18269.455} C_VEL
LIN {X 0,Y 208.22,Z 727.044,A -85,B 0,C 180,E1 -18272.778,E2 -18272.778} C_VEL
LIN {X 0,Y 205.163,Z 736.141,A -85,B 0,C 180,E1 -18276.714,E2 -18276.714} C_VEL
LIN {X 0,Y 202.885,Z 743.192,A -85,B 0,C 180,E1 -18280.79,E2 -18280.79} C_VEL
LIN {X 0,Y 201.304,Z 748.755,A -85,B 0,C 180,E1 -18285.259,E2 -18285.259} C_VEL
LIN {X 0,Y 200.54,Z 752.289,A -85,B 0,C 180,E1 -18289.551,E2 -18289.551} C_VEL
LIN {X 0,Y 200.289,Z 754.29,A -85,B 0,C 180,E1 -18294.16,E2 -18294.16} C_VEL
LIN {X 0,Y 200.442,Z 754.618,A -85,B 0,C 180,E1 -18298.608,E2 -18298.608} C_VEL
LIN {X 0,Y 201.12,Z 753.254,A -85,B 0,C 180,E1 -18303.148,E2 -18303.148} C_VEL
LIN {X 0,Y 202.668,Z 750.003,A -85,B 0,C 180,E1 -18307.873,E2 -18307.873} C_VEL
LIN {X 0,Y 205.095,Z 745.048,A -85,B 0,C 180,E1 -18312.276,E2 -18312.276} C_VEL
LIN {X 0,Y 208.385,Z 738.359,A -85,B 0,C 180,E1 -18316.424,E2 -18316.424} C_VEL
LIN {X 0,Y 212.29,Z 730.165,A -85,B 0,C 180,E1 -18320.166,E2 -18320.166} C_VEL
LIN {X 0,Y 216.951,Z 719.717,A -85,B 0,C 180,E1 -18323.751,E2 -18323.751} C_VEL
LIN {X 0,Y 221.429,Z 708.663,A -85,B 0,C 180,E1 -18326.647,E2 -18326.647} C_VEL
LIN {X 0,Y 226.107,Z 695.641,A -85,B 0,C 180,E1 -18329.276,E2 -18329.276} C_VEL
LIN {X 0,Y 230.179,Z 682.341,A -85,B 0,C 180,E1 -18331.33,E2 -18331.33} C_VEL
LIN {X 0,Y 233.865,Z 667.618,A -85,B 0,C 180,E1 -18333.05,E2 -18333.05} C_VEL
LIN {X 0,Y 236.815,Z 652.159,A -85,B 0,C 180,E1 -18334.373,E2 -18334.373} C_VEL
LIN {X 0,Y 239.007,Z 635.152,A -85,B 0,C 180,E1 -18335.356,E2 -18335.356} C_VEL
LIN {X 0,Y 241.126,Z 604.366,A -85,B 0,C 180,E1 -18336.337,E2 -18336.337} C_VEL
LIN {X 0,Y 243.739,Z 565.021,A -85,B 0,C 180,E1 -18337.467,E2 -18337.467} C_VEL
LIN {X 0,Y 243.595,Z 557.435,A -85,B 0,C 180,E1 -18337.857,E2 -18337.857} C_VEL
LIN {X 0,Y 240.925,Z 537.597,A -85,B 0,C 180,E1 -18339.544,E2 -18339.544} C_VEL
LIN {X 0,Y 240.921,Z 531.076,A -85,B 0,C 180,E1 -18339.865,E2 -18339.865} C_VEL
LIN {X 0,Y 241.844,Z 516.339,A -85,B 0,C 180,E1 -18340.332,E2 -18340.332} C_VEL
LIN {X 0,Y 240.7,Z 488.445,A -85,B 0,C 180,E1 -18342.191,E2 -18342.191} C_VEL
LIN {X 0,Y 250.037,Z 441.986,A -85,B 0,C 180,E1 -18347.763,E2 -18347.763} C_VEL
LIN {X 0,Y 255.466,Z 416.113,A -85,B 0,C 180,E1 -18350.879,E2 -18350.879} C_VEL
LIN {X 0,Y 253.561,Z 406.795,A -85,B 0,C 180,E1 -18353.66,E2 -18353.66} C_VEL
LIN {X 0,Y 251.505,Z 398.358,A -85,B 0,C 180,E1 -18356.809,E2 -18356.809} C_VEL
LIN {X 0,Y 249.659,Z 392.262,A -85,B 0,C 180,E1 -18359.54,E2 -18359.54} C_VEL
LIN {X 0,Y 247.923,Z 386.935,A -85,B 0,C 180,E1 -18362.542,E2 -18362.542} C_VEL
LIN {X 0,Y 246.785,Z 383.748,A -85,B 0,C 180,E1 -18364.71,E2 -18364.71} C_VEL
LIN {X 0,Y 245.723,Z 380.287,A -85,B 0,C 180,E1 -18367.716,E2 -18367.716} C_VEL
LIN {X 0,Y 244.853,Z 376.48,A -85,B 0,C 180,E1 -18372.605,E2 -18372.605} C_VEL
LIN {X 0,Y 244.907,Z 376.153,A -85,B 0,C 180,E1 -18377.829,E2 -18377.829} C_VEL
LIN {X 0,Y 245.38,Z 376.711,A -85,B 0,C 180,E1 -18380.015,E2 -18380.015} C_VEL
LIN {X 0,Y 244.426,Z 383.414,A -85,B 0,C 180,E1 -18382.613,E2 -18382.613} C_VEL
LIN {X 0,Y 244.13,Z 391.988,A -85,B 0,C 180,E1 -18385.636,E2 -18385.636} C_VEL
LIN {X 0,Y 256.154,Z 413.953,A -85,B 0,C 180,E1 -18389.685,E2 -18389.685} C_VEL
LIN {X 0,Y 259.576,Z 420.766,A -85,B 0,C 180,E1 -18390.778,E2 -18390.778} C_VEL
LIN {X 0,Y 240.85,Z 575.105,A -85,B 0,C 180,E1 -18396.732,E2 -18396.732} C_VEL
LIN {X 0,Y 237.142,Z 597.038,A -85,B 0,C 180,E1 -18397.993,E2 -18397.993} C_VEL
LIN {X 0,Y 232.859,Z 617.623,A -85,B 0,C 180,E1 -18399.584,E2 -18399.584} C_VEL
LIN {X 0,Y 227.952,Z 637.756,A -85,B 0,C 180,E1 -18401.6,E2 -18401.6} C_VEL
LIN {X 0,Y 222.617,Z 657.151,A -85,B 0,C 180,E1 -18404.064,E2 -18404.064} C_VEL
LIN {X 0,Y 217.694,Z 673.964,A -85,B 0,C 180,E1 -18406.639,E2 -18406.639} C_VEL
LIN {X 0,Y 215.623,Z 686.451,A -85,B 0,C 180,E1 -18408.112,E2 -18408.112} C_VEL
LIN {X 0,Y 212.767,Z 699.832,A -85,B 0,C 180,E1 -18410.104,E2 -18410.104} C_VEL
LIN {X 0,Y 209.322,Z 713.417,A -85,B 0,C 180,E1 -18412.658,E2 -18412.658} C_VEL
LIN {X 0,Y 205.805,Z 725.58,A -85,B 0,C 180,E1 -18415.533,E2 -18415.533} C_VEL
LIN {X 0,Y 202.091,Z 737.226,A -85,B 0,C 180,E1 -18419.037,E2 -18419.037} C_VEL
LIN {X 0,Y 198.744,Z 747.446,A -85,B 0,C 180,E1 -18422.93,E2 -18422.93} C_VEL
LIN {X 0,Y 195.945,Z 756.03,A -85,B 0,C 180,E1 -18427.186,E2 -18427.186} C_VEL
LIN {X 0,Y 193.809,Z 763.358,A -85,B 0,C 180,E1 -18431.972,E2 -18431.972} C_VEL
LIN {X 0,Y 192.593,Z 768.562,A -85,B 0,C 180,E1 -18436.799,E2 -18436.799} C_VEL
LIN {X 0,Y 192.193,Z 771.943,A -85,B 0,C 180,E1 -18441.628,E2 -18441.628} C_VEL
LIN {X 0,Y 192.239,Z 773.475,A -85,B 0,C 180,E1 -18446.126,E2 -18446.126} C_VEL
LIN {X 0,Y 192.346,Z 773.473,A -85,B 0,C 180,E1 -18450.301,E2 -18450.301} C_VEL
LIN {X 0,Y 192.27,Z 772.058,A -85,B 0,C 180,E1 -18455.075,E2 -18455.075} C_VEL
LIN {X 0,Y 192.224,Z 772.198,A -85,B 0,C 180,E1 -18460.493,E2 -18460.493} C_VEL
LIN {X 0,Y 193.382,Z 770.706,A -85,B 0,C 180,E1 -18466.834,E2 -18466.834} C_VEL
LIN {X 0,Y 196.793,Z 767.238,A -85,B 0,C 180,E1 -18473.668,E2 -18473.668} C_VEL
LIN {X 0,Y 203.171,Z 761.676,A -85,B 0,C 180,E1 -18480.548,E2 -18480.548} C_VEL
LIN {X 0,Y 212.672,Z 754.195,A -85,B 0,C 180,E1 -18487.001,E2 -18487.001} C_VEL
LIN {X 0,Y 225.796,Z 744.608,A -85,B 0,C 180,E1 -18492.998,E2 -18492.998} C_VEL
LIN {X 0,Y 241.244,Z 734.039,A -85,B 0,C 180,E1 -18497.895,E2 -18497.895} C_VEL
LIN {X 0,Y 225.686,Z 742.38,A -85,B 0,C 180,E1 -18502.95,E2 -18502.95} C_VEL
LIN {X 0,Y 213.353,Z 748.778,A -85,B 0,C 180,E1 -18508.656,E2 -18508.656} C_VEL
LIN {X 0,Y 204.56,Z 753.017,A -85,B 0,C 180,E1 -18514.525,E2 -18514.525} C_VEL
LIN {X 0,Y 198.496,Z 755.406,A -85,B 0,C 180,E1 -18520.583,E2 -18520.583} C_VEL
LIN {X 0,Y 194.792,Z 756.034,A -85,B 0,C 180,E1 -18526.646,E2 -18526.646} C_VEL
LIN {X 0,Y 192.941,Z 755.001,A -85,B 0,C 180,E1 -18532.557,E2 -18532.557} C_VEL
LIN {X 0,Y 192.292,Z 752.428,A -85,B 0,C 180,E1 -18538.213,E2 -18538.213} C_VEL
LIN {X 0,Y 192.181,Z 748.624,A -85,B 0,C 180,E1 -18543.282,E2 -18543.282} C_VEL
LIN {X 0,Y 192.446,Z 743.289,A -85,B 0,C 180,E1 -18548.366,E2 -18548.366} C_VEL
LIN {X 0,Y 193.352,Z 736.135,A -85,B 0,C 180,E1 -18553.536,E2 -18553.536} C_VEL
LIN {X 0,Y 195.109,Z 727.288,A -85,B 0,C 180,E1 -18558.541,E2 -18558.541} C_VEL
LIN {X 0,Y 197.716,Z 716.934,A -85,B 0,C 180,E1 -18563.233,E2 -18563.233} C_VEL
LIN {X 0,Y 201.376,Z 704.175,A -85,B 0,C 180,E1 -18567.892,E2 -18567.892} C_VEL
LIN {X 0,Y 205.781,Z 689.734,A -85,B 0,C 180,E1 -18572.141,E2 -18572.141} C_VEL
LIN {X 0,Y 210.635,Z 673.908,A -85,B 0,C 180,E1 -18575.892,E2 -18575.892} C_VEL
LIN {X 0,Y 215.813,Z 656.319,A -85,B 0,C 180,E1 -18579.229,E2 -18579.229} C_VEL
LIN {X 0,Y 220.935,Z 637.705,A -85,B 0,C 180,E1 -18582.052,E2 -18582.052} C_VEL
LIN {X 0,Y 226.04,Z 617.124,A -85,B 0,C 180,E1 -18584.517,E2 -18584.517} C_VEL
LIN {X 0,Y 230.622,Z 595.825,A -85,B 0,C 180,E1 -18586.479,E2 -18586.479} C_VEL
LIN {X 0,Y 234.452,Z 574.128,A -85,B 0,C 180,E1 -18587.962,E2 -18587.962} C_VEL
LIN {X 0,Y 237.854,Z 548.874,A -85,B 0,C 180,E1 -18589.184,E2 -18589.184} C_VEL
LIN {X 0,Y 253.965,Z 419.148,A -85,B 0,C 180,E1 -18594.428,E2 -18594.428} C_VEL
LIN {X 0,Y 242.771,Z 396.87,A -85,B 0,C 180,E1 -18598.287,E2 -18598.287} C_VEL
LIN {X 0,Y 239.518,Z 397.687,A -85,B 0,C 180,E1 -18598.992,E2 -18598.992} C_VEL
LIN {X 0,Y 238.848,Z 398.328,A -85,B 0,C 180,E1 -18599.461,E2 -18599.461} C_VEL
LIN {X 0,Y 241.301,Z 407.722,A -85,B 0,C 180,E1 -18601.735,E2 -18601.735} C_VEL
LIN {X 0,Y 234.149,Z 448.676,A -85,B 0,C 180,E1 -18606.732,E2 -18606.732} C_VEL
LIN {X 0,Y 227.855,Z 487.355,A -85,B 0,C 180,E1 -18611.48,E2 -18611.48} C_VEL
LIN {X 0,Y 229.331,Z 516.378,A -85,B 0,C 180,E1 -18612.993,E2 -18612.993} C_VEL
LIN {X 0,Y 222.519,Z 632.315,A -85,B 0,C 180,E1 -18616.543,E2 -18616.543} C_VEL
LIN {X 0,Y 220.721,Z 648.894,A -85,B 0,C 180,E1 -18617.522,E2 -18617.522} C_VEL
LIN {X 0,Y 218.223,Z 664.643,A -85,B 0,C 180,E1 -18618.902,E2 -18618.902} C_VEL
LIN {X 0,Y 214.997,Z 679.863,A -85,B 0,C 180,E1 -18620.764,E2 -18620.764} C_VEL
LIN {X 0,Y 211.551,Z 693.391,A -85,B 0,C 180,E1 -18622.939,E2 -18622.939} C_VEL
LIN {X 0,Y 207.8,Z 706.031,A -85,B 0,C 180,E1 -18625.582,E2 -18625.582} C_VEL
LIN {X 0,Y 204.028,Z 717.672,A -85,B 0,C 180,E1 -18628.702,E2 -18628.702} C_VEL
LIN {X 0,Y 200.441,Z 727.963,A -85,B 0,C 180,E1 -18632.284,E2 -18632.284} C_VEL
LIN {X 0,Y 197.253,Z 737.027,A -85,B 0,C 180,E1 -18636.399,E2 -18636.399} C_VEL
LIN {X 0,Y 194.901,Z 743.942,A -85,B 0,C 180,E1 -18640.639,E2 -18640.639} C_VEL
LIN {X 0,Y 193.286,Z 749.42,A -85,B 0,C 180,E1 -18645.293,E2 -18645.293} C_VEL
LIN {X 0,Y 192.494,Z 752.984,A -85,B 0,C 180,E1 -18650.045,E2 -18650.045} C_VEL
LIN {X 0,Y 192.297,Z 754.839,A -85,B 0,C 180,E1 -18654.904,E2 -18654.904} C_VEL
LIN {X 0,Y 192.54,Z 754.923,A -85,B 0,C 180,E1 -18659.556,E2 -18659.556} C_VEL
LIN {X 0,Y 193.497,Z 753.171,A -85,B 0,C 180,E1 -18664.635,E2 -18664.635} C_VEL
LIN {X 0,Y 195.34,Z 749.675,A -85,B 0,C 180,E1 -18669.383,E2 -18669.383} C_VEL
LIN {X 0,Y 198.286,Z 744.167,A -85,B 0,C 180,E1 -18674.091,E2 -18674.091} C_VEL
LIN {X 0,Y 201.718,Z 737.65,A -85,B 0,C 180,E1 -18678.026,E2 -18678.026} C_VEL
LIN {X 0,Y 206.171,Z 728.807,A -85,B 0,C 180,E1 -18681.981,E2 -18681.981} C_VEL
LIN {X 0,Y 210.775,Z 719.016,A -85,B 0,C 180,E1 -18685.301,E2 -18685.301} C_VEL
LIN {X 0,Y 215.555,Z 707.71,A -85,B 0,C 180,E1 -18688.234,E2 -18688.234} C_VEL
LIN {X 0,Y 220.306,Z 694.992,A -85,B 0,C 180,E1 -18690.785,E2 -18690.785} C_VEL
LIN {X 0,Y 224.649,Z 681.173,A -85,B 0,C 180,E1 -18692.885,E2 -18692.885} C_VEL
LIN {X 0,Y 228.503,Z 666.193,A -85,B 0,C 180,E1 -18694.606,E2 -18694.606} C_VEL
LIN {X 0,Y 231.581,Z 649.983,A -85,B 0,C 180,E1 -18695.937,E2 -18695.937} C_VEL
LIN {X 0,Y 233.632,Z 633.881,A -85,B 0,C 180,E1 -18696.826,E2 -18696.826} C_VEL
LIN {X 0,Y 240.921,Z 531.076,A -85,B 0,C 180,E1 -18699.865,E2 -18699.865} C_VEL
LIN {X 0,Y 240.831,Z 524.602,A -85,B 0,C 180,E1 -18700.217,E2 -18700.217} C_VEL
LIN {X 0,Y 239.292,Z 515.474,A -85,B 0,C 180,E1 -18701.157,E2 -18701.157} C_VEL
LIN {X 0,Y 236.64,Z 502.462,A -85,B 0,C 180,E1 -18702.717,E2 -18702.717} C_VEL
LIN {X 0,Y 236.253,Z 498.21,A -85,B 0,C 180,E1 -18703.084,E2 -18703.084} C_VEL
LIN {X 0,Y 236.001,Z 488.293,A -85,B 0,C 180,E1 -18703.849,E2 -18703.849} C_VEL
LIN {X 0,Y 245.63,Z 442.94,A -85,B 0,C 180,E1 -18709.326,E2 -18709.326} C_VEL
LIN {X 0,Y 250.545,Z 420.117,A -85,B 0,C 180,E1 -18712.085,E2 -18712.085} C_VEL
LIN {X 0,Y 249.035,Z 411.206,A -85,B 0,C 180,E1 -18714.932,E2 -18714.932} C_VEL
LIN {X 0,Y 246.991,Z 402.953,A -85,B 0,C 180,E1 -18718.143,E2 -18718.143} C_VEL
LIN {X 0,Y 245.242,Z 396.209,A -85,B 0,C 180,E1 -18721.635,E2 -18721.635} C_VEL
LIN {X 0,Y 243.632,Z 391.048,A -85,B 0,C 180,E1 -18724.943,E2 -18724.943} C_VEL
LIN {X 0,Y 242.651,Z 387.553,A -85,B 0,C 180,E1 -18728.053,E2 -18728.053} C_VEL
LIN {X 0,Y 242.095,Z 384.318,A -85,B 0,C 180,E1 -18732.159,E2 -18732.159} C_VEL
LIN {X 0,Y 241.773,Z 383.578,A -85,B 0,C 180,E1 -18735.593,E2 -18735.593} C_VEL
LIN {X 0,Y 242.607,Z 384.034,A -85,B 0,C 180,E1 -18739.5,E2 -18739.5} C_VEL
LIN {X 0,Y 240.796,Z 398.417,A -85,B 0,C 180,E1 -18744.795,E2 -18744.795} C_VEL
LIN {X 0,Y 241.096,Z 400.768,A -85,B 0,C 180,E1 -18745.549,E2 -18745.549} C_VEL
LIN {X 0,Y 252.977,Z 422.935,A -85,B 0,C 180,E1 -18749.606,E2 -18749.606} C_VEL
LIN {X 0,Y 253.143,Z 424.148,A -85,B 0,C 180,E1 -18749.716,E2 -18749.716} C_VEL
LIN {X 0,Y 234.137,Z 574.847,A -85,B 0,C 180,E1 -18755.683,E2 -18755.683} C_VEL
LIN {X 0,Y 230.288,Z 596.905,A -85,B 0,C 180,E1 -18756.982,E2 -18756.982} C_VEL
LIN {X 0,Y 225.829,Z 617.631,A -85,B 0,C 180,E1 -18758.628,E2 -18758.628} C_VEL
LIN {X 0,Y 220.735,Z 637.855,A -85,B 0,C 180,E1 -18760.712,E2 -18760.712} C_VEL
LIN {X 0,Y 215.08,Z 657.785,A -85,B 0,C 180,E1 -18763.325,E2 -18763.325} C_VEL
LIN {X 0,Y 213.95,Z 662.473,A -85,B 0,C 180,E1 -18763.88,E2 -18763.88} C_VEL
LIN {X 0,Y 212.068,Z 675.752,A -85,B 0,C 180,E1 -18765.186,E2 -18765.186} C_VEL
LIN {X 0,Y 209.383,Z 689.628,A -85,B 0,C 180,E1 -18766.937,E2 -18766.937} C_VEL
LIN {X 0,Y 206.141,Z 703.112,A -85,B 0,C 180,E1 -18769.1,E2 -18769.1} C_VEL
LIN {X 0,Y 202.618,Z 715.323,A -85,B 0,C 180,E1 -18771.559,E2 -18771.559} C_VEL
LIN {X 0,Y 198.504,Z 727.958,A -85,B 0,C 180,E1 -18774.783,E2 -18774.783} C_VEL
LIN {X 0,Y 194.577,Z 739.128,A -85,B 0,C 180,E1 -18778.394,E2 -18778.394} C_VEL
LIN {X 0,Y 190.917,Z 749.082,A -85,B 0,C 180,E1 -18782.561,E2 -18782.561} C_VEL
LIN {X 0,Y 187.905,Z 757.538,A -85,B 0,C 180,E1 -18787.147,E2 -18787.147} C_VEL
LIN {X 0,Y 185.717,Z 764.291,A -85,B 0,C 180,E1 -18792.133,E2 -18792.133} C_VEL
LIN {X 0,Y 184.529,Z 769.111,A -85,B 0,C 180,E1 -18797.168,E2 -18797.168} C_VEL
LIN {X 0,Y 184.184,Z 772.034,A -85,B 0,C 180,E1 -18802.204,E2 -18802.204} C_VEL
LIN {X 0,Y 184.272,Z 773.191,A -85,B 0,C 180,E1 -18806.893,E2 -18806.893} C_VEL
LIN {X 0,Y 184.351,Z 772.849,A -85,B 0,C 180,E1 -18811.246,E2 -18811.246} C_VEL
LIN {X 0,Y 184.284,Z 771.346,A -85,B 0,C 180,E1 -18815.608,E2 -18815.608} C_VEL
LIN {X 0,Y 184.326,Z 771.567,A -85,B 0,C 180,E1 -18821.581,E2 -18821.581} C_VEL
LIN {X 0,Y 185.928,Z 770.111,A -85,B 0,C 180,E1 -18828.502,E2 -18828.502} C_VEL
LIN {X 0,Y 190.02,Z 766.792,A -85,B 0,C 180,E1 -18835.564,E2 -18835.564} C_VEL
LIN {X 0,Y 197.547,Z 761.296,A -85,B 0,C 180,E1 -18842.794,E2 -18842.794} C_VEL
LIN {X 0,Y 208.757,Z 753.751,A -85,B 0,C 180,E1 -18849.573,E2 -18849.573} C_VEL
LIN {X 0,Y 223.785,Z 744.252,A -85,B 0,C 180,E1 -18855.636,E2 -18855.636} C_VEL
LIN {X 0,Y 231.299,Z 739.685,A -85,B 0,C 180,E1 -18857.973,E2 -18857.973} C_VEL
LIN {X 0,Y 216.082,Z 746.688,A -85,B 0,C 180,E1 -18863.183,E2 -18863.183} C_VEL
LIN {X 0,Y 204.094,Z 751.883,A -85,B 0,C 180,E1 -18869.044,E2 -18869.044} C_VEL
LIN {X 0,Y 195.135,Z 755.238,A -85,B 0,C 180,E1 -18875.479,E2 -18875.479} C_VEL
LIN {X 0,Y 189.422,Z 756.643,A -85,B 0,C 180,E1 -18881.856,E2 -18881.856} C_VEL
LIN {X 0,Y 186.113,Z 756.324,A -85,B 0,C 180,E1 -18888.221,E2 -18888.221} C_VEL
LIN {X 0,Y 184.625,Z 754.377,A -85,B 0,C 180,E1 -18894.407,E2 -18894.407} C_VEL
LIN {X 0,Y 184.224,Z 751.132,A -85,B 0,C 180,E1 -18900.001,E2 -18900.001} C_VEL
LIN {X 0,Y 184.231,Z 746.534,A -85,B 0,C 180,E1 -18905.295,E2 -18905.295} C_VEL
LIN {X 0,Y 184.735,Z 740.339,A -85,B 0,C 180,E1 -18910.605,E2 -18910.605} C_VEL
LIN {X 0,Y 186.028,Z 732.351,A -85,B 0,C 180,E1 -18915.91,E2 -18915.91} C_VEL
LIN {X 0,Y 188.336,Z 722.351,A -85,B 0,C 180,E1 -18921.163,E2 -18921.163} C_VEL
LIN {X 0,Y 191.548,Z 710.819,A -85,B 0,C 180,E1 -18926.008,E2 -18926.008} C_VEL
LIN {X 0,Y 195.517,Z 697.858,A -85,B 0,C 180,E1 -18930.418,E2 -18930.418} C_VEL
LIN {X 0,Y 200.217,Z 683.004,A -85,B 0,C 180,E1 -18934.51,E2 -18934.51} C_VEL
LIN {X 0,Y 205.401,Z 666.436,A -85,B 0,C 180,E1 -18938.187,E2 -18938.187} C_VEL
LIN {X 0,Y 210.593,Z 648.943,A -85,B 0,C 180,E1 -18941.297,E2 -18941.297} C_VEL
LIN {X 0,Y 215.838,Z 629.725,A -85,B 0,C 180,E1 -18944.018,E2 -18944.018} C_VEL
LIN {X 0,Y 220.744,Z 609.527,A -85,B 0,C 180,E1 -18946.259,E2 -18946.259} C_VEL
LIN {X 0,Y 225.138,Z 588.374,A -85,B 0,C 180,E1 -18948.065,E2 -18948.065} C_VEL
LIN {X 0,Y 228.911,Z 566.276,A -85,B 0,C 180,E1 -18949.454,E2 -18949.454} C_VEL
LIN {X 0,Y 247.588,Z 422.026,A -85,B 0,C 180,E1 -18955.531,E2 -18955.531} C_VEL
LIN {X 0,Y 239.359,Z 405.458,A -85,B 0,C 180,E1 -18958.449,E2 -18958.449} C_VEL
LIN {X 0,Y 235.921,Z 406.764,A -85,B 0,C 180,E1 -18959.146,E2 -18959.146} C_VEL
LIN {X 0,Y 234.511,Z 407.098,A -85,B 0,C 180,E1 -18959.65,E2 -18959.65} C_VEL
LIN {X 0,Y 234.955,Z 409.752,A -85,B 0,C 180,E1 -18960.417,E2 -18960.417} C_VEL
LIN {X 0,Y 235.095,Z 411.255,A -85,B 0,C 180,E1 -18960.716,E2 -18960.716} C_VEL
LIN {X 0,Y 227.5,Z 453.154,A -85,B 0,C 180,E1 -18965.872,E2 -18965.872} C_VEL
LIN {X 0,Y 221.629,Z 487.647,A -85,B 0,C 180,E1 -18970.169,E2 -18970.169} C_VEL
LIN {X 0,Y 223.021,Z 517.149,A -85,B 0,C 180,E1 -18971.754,E2 -18971.754} C_VEL
LIN {X 0,Y 215.918,Z 632.684,A -85,B 0,C 180,E1 -18975.365,E2 -18975.365} C_VEL
LIN {X 0,Y 214.063,Z 649.126,A -85,B 0,C 180,E1 -18976.354,E2 -18976.354} C_VEL
LIN {X 0,Y 211.546,Z 664.466,A -85,B 0,C 180,E1 -18977.717,E2 -18977.717} C_VEL
LIN {X 0,Y 208.401,Z 678.939,A -85,B 0,C 180,E1 -18979.492,E2 -18979.492} C_VEL
LIN {X 0,Y 204.58,Z 693.449,A -85,B 0,C 180,E1 -18981.849,E2 -18981.849} C_VEL
LIN {X 0,Y 200.654,Z 706.168,A -85,B 0,C 180,E1 -18984.564,E2 -18984.564} C_VEL
LIN {X 0,Y 196.817,Z 717.49,A -85,B 0,C 180,E1 -18987.668,E2 -18987.668} C_VEL
LIN {X 0,Y 193.193,Z 727.477,A -85,B 0,C 180,E1 -18991.183,E2 -18991.183} C_VEL
LIN {X 0,Y 189.762,Z 736.705,A -85,B 0,C 180,E1 -18995.439,E2 -18995.439} C_VEL
LIN {X 0,Y 187.211,Z 743.822,A -85,B 0,C 180,E1 -18999.837,E2 -18999.837} C_VEL
LIN {X 0,Y 185.431,Z 749.427,A -85,B 0,C 180,E1 -19004.677,E2 -19004.677} C_VEL
LIN {X 0,Y 184.556,Z 753.097,A -85,B 0,C 180,E1 -19009.491,E2 -19009.491} C_VEL
LIN {X 0,Y 184.304,Z 755.053,A -85,B 0,C 180,E1 -19014.346,E2 -19014.346} C_VEL
LIN {X 0,Y 184.518,Z 755.416,A -85,B 0,C 180,E1 -19019.256,E2 -19019.256} C_VEL
LIN {X 0,Y 185.354,Z 754.108,A -85,B 0,C 180,E1 -19024.121,E2 -19024.121} C_VEL
LIN {X 0,Y 187.315,Z 750.745,A -85,B 0,C 180,E1 -19029.43,E2 -19029.43} C_VEL
LIN {X 0,Y 190.067,Z 746.008,A -85,B 0,C 180,E1 -19033.974,E2 -19033.974} C_VEL
LIN {X 0,Y 193.851,Z 739.381,A -85,B 0,C 180,E1 -19038.402,E2 -19038.402} C_VEL
LIN {X 0,Y 198.337,Z 731.178,A -85,B 0,C 180,E1 -19042.41,E2 -19042.41} C_VEL
LIN {X 0,Y 203.498,Z 720.941,A -85,B 0,C 180,E1 -19046.129,E2 -19046.129} C_VEL
LIN {X 0,Y 208.473,Z 710.061,A -85,B 0,C 180,E1 -19049.142,E2 -19049.142} C_VEL
LIN {X 0,Y 213.673,Z 697.07,A -85,B 0,C 180,E1 -19051.885,E2 -19051.885} C_VEL
LIN {X 0,Y 218.087,Z 684.209,A -85,B 0,C 180,E1 -19053.966,E2 -19053.966} C_VEL
LIN {X 0,Y 222.153,Z 669.621,A -85,B 0,C 180,E1 -19055.745,E2 -19055.745} C_VEL
LIN {X 0,Y 225.402,Z 654.619,A -85,B 0,C 180,E1 -19057.1,E2 -19057.1} C_VEL
LIN {X 0,Y 227.847,Z 638.125,A -85,B 0,C 180,E1 -19058.116,E2 -19058.116} C_VEL
LIN {X 0,Y 229.488,Z 618.664,A -85,B 0,C 180,E1 -19058.827,E2 -19058.827} C_VEL
LIN {X 0,Y 236.881,Z 517.514,A -85,B 0,C 180,E1 -19061.814,E2 -19061.814} C_VEL
LIN {X 0,Y 236.253,Z 498.21,A -85,B 0,C 180,E1 -19063.084,E2 -19063.084} C_VEL
LIN {X 0,Y 235.789,Z 492.147,A -85,B 0,C 180,E1 -19063.734,E2 -19063.734} C_VEL
LIN {X 0,Y 234.909,Z 483.19,A -85,B 0,C 180,E1 -19065.343,E2 -19065.343} C_VEL
LIN {X 0,Y 235.06,Z 473.605,A -85,B 0,C 180,E1 -19067.251,E2 -19067.251} C_VEL
LIN {X 0,Y 235.804,Z 468.863,A -85,B 0,C 180,E1 -19067.948,E2 -19067.948} C_VEL
LIN {X 0,Y 244.907,Z 428.771,A -85,B 0,C 180,E1 -19072.755,E2 -19072.755} C_VEL
LIN {X 0,Y 245.888,Z 424.258,A -85,B 0,C 180,E1 -19073.344,E2 -19073.344} C_VEL
LIN {X 0,Y 244.59,Z 415.72,A -85,B 0,C 180,E1 -19076.249,E2 -19076.249} C_VEL
LIN {X 0,Y 242.963,Z 408.393,A -85,B 0,C 180,E1 -19079.292,E2 -19079.292} C_VEL
LIN {X 0,Y 241.482,Z 402.215,A -85,B 0,C 180,E1 -19082.61,E2 -19082.61} C_VEL
LIN {X 0,Y 240.315,Z 397.785,A -85,B 0,C 180,E1 -19085.73,E2 -19085.73} C_VEL
LIN {X 0,Y 239.562,Z 394.77,A -85,B 0,C 180,E1 -19088.465,E2 -19088.465} C_VEL
LIN {X 0,Y 239.246,Z 391.417,A -85,B 0,C 180,E1 -19093.042,E2 -19093.042} C_VEL
LIN {X 0,Y 239.377,Z 391.156,A -85,B 0,C 180,E1 -19097.25,E2 -19097.25} C_VEL
LIN {X 0,Y 239.809,Z 391.49,A -85,B 0,C 180,E1 -19098.978,E2 -19098.978} C_VEL
LIN {X 0,Y 237.902,Z 404.084,A -85,B 0,C 180,E1 -19103.63,E2 -19103.63} C_VEL
LIN {X 0,Y 237.833,Z 409.265,A -85,B 0,C 180,E1 -19105.391,E2 -19105.391} C_VEL
LIN {X 0,Y 246.865,Z 426.525,A -85,B 0,C 180,E1 -19108.579,E2 -19108.579} C_VEL
LIN {X 0,Y 227.363,Z 575.096,A -85,B 0,C 180,E1 -19114.624,E2 -19114.624} C_VEL
LIN {X 0,Y 223.471,Z 596.678,A -85,B 0,C 180,E1 -19115.926,E2 -19115.926} C_VEL
LIN {X 0,Y 218.919,Z 617.233,A -85,B 0,C 180,E1 -19117.594,E2 -19117.594} C_VEL
LIN {X 0,Y 213.463,Z 638.211,A -85,B 0,C 180,E1 -19119.815,E2 -19119.815} C_VEL
LIN {X 0,Y 210.519,Z 649.065,A -85,B 0,C 180,E1 -19121.12,E2 -19121.12} C_VEL
LIN {X 0,Y 209.323,Z 660.622,A -85,B 0,C 180,E1 -19121.968,E2 -19121.968} C_VEL
LIN {X 0,Y 207.267,Z 674.027,A -85,B 0,C 180,E1 -19123.251,E2 -19123.251} C_VEL
LIN {X 0,Y 204.336,Z 688.148,A -85,B 0,C 180,E1 -19125.008,E2 -19125.008} C_VEL
LIN {X 0,Y 200.782,Z 701.77,A -85,B 0,C 180,E1 -19127.181,E2 -19127.181} C_VEL
LIN {X 0,Y 196.558,Z 715.349,A -85,B 0,C 180,E1 -19129.953,E2 -19129.953} C_VEL
LIN {X 0,Y 192.018,Z 728.138,A -85,B 0,C 180,E1 -19133.31,E2 -19133.31} C_VEL
LIN {X 0,Y 187.669,Z 739.331,A -85,B 0,C 180,E1 -19137.087,E2 -19137.087} C_VEL
LIN {X 0,Y 183.446,Z 749.807,A -85,B 0,C 180,E1 -19141.698,E2 -19141.698} C_VEL
LIN {X 0,Y 180.379,Z 757.492,A -85,B 0,C 180,E1 -19146.148,E2 -19146.148} C_VEL
LIN {X 0,Y 177.966,Z 764.139,A -85,B 0,C 180,E1 -19151.326,E2 -19151.326} C_VEL
LIN {X 0,Y 176.611,Z 768.858,A -85,B 0,C 180,E1 -19156.582,E2 -19156.582} C_VEL
LIN {X 0,Y 176.192,Z 771.712,A -85,B 0,C 180,E1 -19161.848,E2 -19161.848} C_VEL
LIN {X 0,Y 176.275,Z 772.814,A -85,B 0,C 180,E1 -19166.752,E2 -19166.752} C_VEL
LIN {X 0,Y 176.365,Z 772.479,A -85,B 0,C 180,E1 -19170.978,E2 -19170.978} C_VEL
LIN {X 0,Y 176.306,Z 770.772,A -85,B 0,C 180,E1 -19175.536,E2 -19175.536} C_VEL
LIN {X 0,Y 176.266,Z 770.679,A -85,B 0,C 180,E1 -19176.946,E2 -19176.946} C_VEL
LIN {X 0,Y 176.557,Z 770.88,A -85,B 0,C 180,E1 -19183.429,E2 -19183.429} C_VEL
LIN {X 0,Y 178.944,Z 769.314,A -85,B 0,C 180,E1 -19190.957,E2 -19190.957} C_VEL
LIN {X 0,Y 184.319,Z 765.832,A -85,B 0,C 180,E1 -19198.517,E2 -19198.517} C_VEL
LIN {X 0,Y 193.219,Z 760.434,A -85,B 0,C 180,E1 -19205.788,E2 -19205.788} C_VEL
LIN {X 0,Y 206.444,Z 752.847,A -85,B 0,C 180,E1 -19212.695,E2 -19212.695} C_VEL
LIN {X 0,Y 221.301,Z 744.666,A -85,B 0,C 180,E1 -19218.036,E2 -19218.036} C_VEL
LIN {X 0,Y 206.407,Z 750.458,A -85,B 0,C 180,E1 -19223.43,E2 -19223.43} C_VEL
LIN {X 0,Y 194.369,Z 754.651,A -85,B 0,C 180,E1 -19229.728,E2 -19229.728} C_VEL
LIN {X 0,Y 185.725,Z 756.942,A -85,B 0,C 180,E1 -19236.524,E2 -19236.524} C_VEL
LIN {X 0,Y 180.215,Z 757.341,A -85,B 0,C 180,E1 -19243.564,E2 -19243.564} C_VEL
LIN {X 0,Y 177.432,Z 755.995,A -85,B 0,C 180,E1 -19250.268,E2 -19250.268} C_VEL
LIN {X 0,Y 176.405,Z 753.242,A -85,B 0,C 180,E1 -19256.427,E2 -19256.427} C_VEL
LIN {X 0,Y 176.184,Z 749.377,A -85,B 0,C 180,E1 -19261.953,E2 -19261.953} C_VEL
LIN {X 0,Y 176.341,Z 744.31,A -85,B 0,C 180,E1 -19267.167,E2 -19267.167} C_VEL
LIN {X 0,Y 177.132,Z 737.32,A -85,B 0,C 180,E1 -19272.719,E2 -19272.719} C_VEL
LIN {X 0,Y 178.85,Z 728.436,A -85,B 0,C 180,E1 -19278.245,E2 -19278.245} C_VEL
LIN {X 0,Y 181.712,Z 717.415,A -85,B 0,C 180,E1 -19283.684,E2 -19283.684} C_VEL
LIN {X 0,Y 185.523,Z 704.794,A -85,B 0,C 180,E1 -19288.664,E2 -19288.664} C_VEL
LIN {X 0,Y 190.1,Z 690.615,A -85,B 0,C 180,E1 -19293.163,E2 -19293.163} C_VEL
LIN {X 0,Y 195.235,Z 674.865,A -85,B 0,C 180,E1 -19297.181,E2 -19297.181} C_VEL
LIN {X 0,Y 200.721,Z 657.439,A -85,B 0,C 180,E1 -19300.736,E2 -19300.736} C_VEL
LIN {X 0,Y 206.127,Z 639.078,A -85,B 0,C 180,E1 -19303.714,E2 -19303.714} C_VEL
LIN {X 0,Y 211.54,Z 618.674,A -85,B 0,C 180,E1 -19306.318,E2 -19306.318} C_VEL
LIN {X 0,Y 216.227,Z 598.503,A -85,B 0,C 180,E1 -19308.315,E2 -19308.315} C_VEL
LIN {X 0,Y 220.446,Z 576.842,A -85,B 0,C 180,E1 -19309.943,E2 -19309.943} C_VEL
LIN {X 0,Y 223.937,Z 553.777,A -85,B 0,C 180,E1 -19311.17,E2 -19311.17} C_VEL
LIN {X 0,Y 241.283,Z 424.9,A -85,B 0,C 180,E1 -19316.659,E2 -19316.659} C_VEL
LIN {X 0,Y 236.132,Z 414.398,A -85,B 0,C 180,E1 -19318.539,E2 -19318.539} C_VEL
LIN {X 0,Y 234.132,Z 415.034,A -85,B 0,C 180,E1 -19318.956,E2 -19318.956} C_VEL
LIN {X 0,Y 229.579,Z 418.365,A -85,B 0,C 180,E1 -19319.797,E2 -19319.797} C_VEL
LIN {X 0,Y 228.056,Z 420.524,A -85,B 0,C 180,E1 -19320.3,E2 -19320.3} C_VEL
LIN {X 0,Y 220.705,Z 458.49,A -85,B 0,C 180,E1 -19325.079,E2 -19325.079} C_VEL
LIN {X 0,Y 215.516,Z 488.142,A -85,B 0,C 180,E1 -19328.801,E2 -19328.801} C_VEL
LIN {X 0,Y 216.788,Z 517.937,A -85,B 0,C 180,E1 -19330.454,E2 -19330.454} C_VEL
LIN {X 0,Y 209.409,Z 633.039,A -85,B 0,C 180,E1 -19334.116,E2 -19334.116} C_VEL
LIN {X 0,Y 207.455,Z 649.632,A -85,B 0,C 180,E1 -19335.135,E2 -19335.135} C_VEL
LIN {X 0,Y 204.727,Z 665.469,A -85,B 0,C 180,E1 -19336.583,E2 -19336.583} C_VEL
LIN {X 0,Y 201.224,Z 680.683,A -85,B 0,C 180,E1 -19338.533,E2 -19338.533} C_VEL
LIN {X 0,Y 197.526,Z 694.032,A -85,B 0,C 180,E1 -19340.786,E2 -19340.786} C_VEL
LIN {X 0,Y 193.378,Z 706.849,A -85,B 0,C 180,E1 -19343.614,E2 -19343.614} C_VEL
LIN {X 0,Y 189.202,Z 718.602,A -85,B 0,C 180,E1 -19346.967,E2 -19346.967} C_VEL
LIN {X 0,Y 185.15,Z 729.144,A -85,B 0,C 180,E1 -19350.925,E2 -19350.925} C_VEL
LIN {X 0,Y 181.739,Z 737.915,A -85,B 0,C 180,E1 -19355.245,E2 -19355.245} C_VEL
LIN {X 0,Y 179.083,Z 744.968,A -85,B 0,C 180,E1 -19359.963,E2 -19359.963} C_VEL
LIN {X 0,Y 177.326,Z 750.379,A -85,B 0,C 180,E1 -19365.029,E2 -19365.029} C_VEL
LIN {X 0,Y 176.488,Z 753.875,A -85,B 0,C 180,E1 -19370.213,E2 -19370.213} C_VEL
LIN {X 0,Y 176.314,Z 755.598,A -85,B 0,C 180,E1 -19375.166,E2 -19375.166} C_VEL
LIN {X 0,Y 176.634,Z 755.745,A -85,B 0,C 180,E1 -19380.247,E2 -19380.247} C_VEL
LIN {X 0,Y 177.819,Z 754.039,A -85,B 0,C 180,E1 -19385.783,E2 -19385.783} C_VEL
LIN {X 0,Y 180.036,Z 750.598,A -85,B 0,C 180,E1 -19390.947,E2 -19390.947} C_VEL
LIN {X 0,Y 183.467,Z 745.165,A -85,B 0,C 180,E1 -19395.997,E2 -19395.997} C_VEL
LIN {X 0,Y 187.403,Z 738.745,A -85,B 0,C 180,E1 -19400.194,E2 -19400.194} C_VEL
LIN {X 0,Y 192.516,Z 729.865,A -85,B 0,C 180,E1 -19404.429,E2 -19404.429} C_VEL
LIN {X 0,Y 197.708,Z 720.11,A -85,B 0,C 180,E1 -19407.925,E2 -19407.925} C_VEL
LIN {X 0,Y 203.273,Z 708.331,A -85,B 0,C 180,E1 -19411.102,E2 -19411.102} C_VEL
LIN {X 0,Y 208.521,Z 695.65,A -85,B 0,C 180,E1 -19413.715,E2 -19413.715} C_VEL
LIN {X 0,Y 213.551,Z 681.099,A -85,B 0,C 180,E1 -19415.961,E2 -19415.961} C_VEL
LIN {X 0,Y 217.574,Z 666.676,A -85,B 0,C 180,E1 -19417.626,E2 -19417.626} C_VEL
LIN {X 0,Y 220.969,Z 650.242,A -85,B 0,C 180,E1 -19418.984,E2 -19418.984} C_VEL
LIN {X 0,Y 223.162,Z 634.232,A -85,B 0,C 180,E1 -19419.866,E2 -19419.866} C_VEL
LIN {X 0,Y 232.101,Z 518.594,A -85,B 0,C 180,E1 -19423.368,E2 -19423.368} C_VEL
LIN {X 0,Y 231.248,Z 490.16,A -85,B 0,C 180,E1 -19425.36,E2 -19425.36} C_VEL
LIN {X 0,Y 235.804,Z 468.863,A -85,B 0,C 180,E1 -19427.948,E2 -19427.948} C_VEL
LIN {X 0,Y 236.757,Z 462.356,A -85,B 0,C 180,E1 -19428.95,E2 -19428.95} C_VEL
LIN {X 0,Y 237.538,Z 446.235,A -85,B 0,C 180,E1 -19432.301,E2 -19432.301} C_VEL
LIN {X 0,Y 238.558,Z 440.651,A -85,B 0,C 180,E1 -19433.146,E2 -19433.146} C_VEL
LIN {X 0,Y 241.411,Z 428.499,A -85,B 0,C 180,E1 -19434.652,E2 -19434.652} C_VEL
LIN {X 0,Y 240.158,Z 420.19,A -85,B 0,C 180,E1 -19437.628,E2 -19437.628} C_VEL
LIN {X 0,Y 238.913,Z 412.936,A -85,B 0,C 180,E1 -19440.958,E2 -19440.958} C_VEL
LIN {X 0,Y 237.515,Z 407.242,A -85,B 0,C 180,E1 -19444.345,E2 -19444.345} C_VEL
LIN {X 0,Y 236.968,Z 403.964,A -85,B 0,C 180,E1 -19447.028,E2 -19447.028} C_VEL
LIN {X 0,Y 236.536,Z 402.082,A -85,B 0,C 180,E1 -19448.752,E2 -19448.752} C_VEL
LIN {X 0,Y 236.458,Z 398.899,A -85,B 0,C 180,E1 -19453.198,E2 -19453.198} C_VEL
LIN {X 0,Y 236.612,Z 398.663,A -85,B 0,C 180,E1 -19457.263,E2 -19457.263} C_VEL
LIN {X 0,Y 236.919,Z 399.079,A -85,B 0,C 180,E1 -19458.452,E2 -19458.452} C_VEL
LIN {X 0,Y 234.749,Z 412.233,A -85,B 0,C 180,E1 -19463.335,E2 -19463.335} C_VEL
LIN {X 0,Y 234.637,Z 417.994,A -85,B 0,C 180,E1 -19465.272,E2 -19465.272} C_VEL
LIN {X 0,Y 240.528,Z 429.545,A -85,B 0,C 180,E1 -19467.426,E2 -19467.426} C_VEL
LIN {X 0,Y 220.68,Z 574.974,A -85,B 0,C 180,E1 -19473.5,E2 -19473.5} C_VEL
LIN {X 0,Y 216.581,Z 596.883,A -85,B 0,C 180,E1 -19474.862,E2 -19474.862} C_VEL
LIN {X 0,Y 211.761,Z 617.854,A -85,B 0,C 180,E1 -19476.619,E2 -19476.619} C_VEL
LIN {X 0,Y 206.872,Z 636.815,A -85,B 0,C 180,E1 -19478.583,E2 -19478.583} C_VEL
LIN {X 0,Y 206.083,Z 648.541,A -85,B 0,C 180,E1 -19479.236,E2 -19479.236} C_VEL
LIN {X 0,Y 204.581,Z 661.318,A -85,B 0,C 180,E1 -19480.174,E2 -19480.174} C_VEL
LIN {X 0,Y 202.164,Z 675.307,A -85,B 0,C 180,E1 -19481.561,E2 -19481.561} C_VEL
LIN {X 0,Y 198.846,Z 689.587,A -85,B 0,C 180,E1 -19483.404,E2 -19483.404} C_VEL
LIN {X 0,Y 194.793,Z 703.544,A -85,B 0,C 180,E1 -19485.732,E2 -19485.732} C_VEL
LIN {X 0,Y 190.047,Z 717.22,A -85,B 0,C 180,E1 -19488.685,E2 -19488.685} C_VEL
LIN {X 0,Y 185.29,Z 729.33,A -85,B 0,C 180,E1 -19492.041,E2 -19492.041} C_VEL
LIN {X 0,Y 180.544,Z 740.344,A -85,B 0,C 180,E1 -19495.994,E2 -19495.994} C_VEL
LIN {X 0,Y 176.281,Z 749.911,A -85,B 0,C 180,E1 -19500.436,E2 -19500.436} C_VEL
LIN {X 0,Y 172.725,Z 757.893,A -85,B 0,C 180,E1 -19505.372,E2 -19505.372} C_VEL
LIN {X 0,Y 170.117,Z 764.366,A -85,B 0,C 180,E1 -19510.788,E2 -19510.788} C_VEL
LIN {X 0,Y 168.648,Z 768.824,A -85,B 0,C 180,E1 -19516.286,E2 -19516.286} C_VEL
LIN {X 0,Y 168.195,Z 771.522,A -85,B 0,C 180,E1 -19521.801,E2 -19521.801} C_VEL
LIN {X 0,Y 168.288,Z 772.462,A -85,B 0,C 180,E1 -19526.939,E2 -19526.939} C_VEL
LIN {X 0,Y 168.371,Z 771.977,A -85,B 0,C 180,E1 -19531.365,E2 -19531.365} C_VEL
LIN {X 0,Y 168.323,Z 770.081,A -85,B 0,C 180,E1 -19536.142,E2 -19536.142} C_VEL
LIN {X 0,Y 168.303,Z 769.82,A -85,B 0,C 180,E1 -19537.514,E2 -19537.514} C_VEL
LIN {X 0,Y 168.793,Z 770.229,A -85,B 0,C 180,E1 -19544.76,E2 -19544.76} C_VEL
LIN {X 0,Y 171.509,Z 768.983,A -85,B 0,C 180,E1 -19552.271,E2 -19552.271} C_VEL
LIN {X 0,Y 177.821,Z 765.679,A -85,B 0,C 180,E1 -19560.405,E2 -19560.405} C_VEL
LIN {X 0,Y 188.556,Z 760.188,A -85,B 0,C 180,E1 -19568.35,E2 -19568.35} C_VEL
LIN {X 0,Y 203.653,Z 752.741,A -85,B 0,C 180,E1 -19575.393,E2 -19575.393} C_VEL
LIN {X 0,Y 211.316,Z 749.021,A -85,B 0,C 180,E1 -19578.071,E2 -19578.071} C_VEL
LIN {X 0,Y 196.422,Z 753.766,A -85,B 0,C 180,E1 -19583.81,E2 -19583.81} C_VEL
LIN {X 0,Y 184.626,Z 756.871,A -85,B 0,C 180,E1 -19590.475,E2 -19590.475} C_VEL
LIN {X 0,Y 176.34,Z 758.119,A -85,B 0,C 180,E1 -19597.674,E2 -19597.674} C_VEL
LIN {X 0,Y 171.293,Z 757.505,A -85,B 0,C 180,E1 -19605.119,E2 -19605.119} C_VEL
LIN {X 0,Y 168.972,Z 755.218,A -85,B 0,C 180,E1 -19612.179,E2 -19612.179} C_VEL
LIN {X 0,Y 168.29,Z 751.818,A -85,B 0,C 180,E1 -19618.299,E2 -19618.299} C_VEL
LIN {X 0,Y 168.197,Z 747.451,A -85,B 0,C 180,E1 -19623.75,E2 -19623.75} C_VEL
LIN {X 0,Y 168.584,Z 741.268,A -85,B 0,C 180,E1 -19629.56,E2 -19629.56} C_VEL
LIN {X 0,Y 169.788,Z 733.311,A -85,B 0,C 180,E1 -19635.368,E2 -19635.368} C_VEL
LIN {X 0,Y 172.098,Z 723.356,A -85,B 0,C 180,E1 -19641.114,E2 -19641.114} C_VEL
LIN {X 0,Y 175.56,Z 711.417,A -85,B 0,C 180,E1 -19646.594,E2 -19646.594} C_VEL
LIN {X 0,Y 179.882,Z 698.076,A -85,B 0,C 180,E1 -19651.501,E2 -19651.501} C_VEL
LIN {X 0,Y 184.919,Z 683.09,A -85,B 0,C 180,E1 -19655.922,E2 -19655.922} C_VEL
LIN {X 0,Y 190.431,Z 666.536,A -85,B 0,C 180,E1 -19659.835,E2 -19659.835} C_VEL
